      end
      $ 545 "Wait: 0.3"
      sleep(0.3)
      $ 546 "Set CO[1]=Encender"
      set_configurable_digital_out(1, True)
      $ 547 "Wait: 0.3"
      sleep(0.3)
      $ 548 "Loop 1 times"
      Loop_85 = 0
      while (Loop_85 < 1):
        $ 549 "bajar≔pose_add(get_actual_tcp_pose(), bajada_broca)"
        global bajar= pose_add ( get_actual_tcp_pose (), bajada_broca)
        $ 550 "bajar" "breakAfter"
        movel(bajar, a=0.005, v=0.001)
        $ 551 "subir≔pose_sub(get_actual_tcp_pose(), bajada_broca)"
        global subir= pose_sub ( get_actual_tcp_pose (), bajada_broca)
        $ 552 "subir" "breakAfter"
        movel(subir, a=0.01, v=0.005)
        $ 553 "bajada_broca≔pose_sub(bajada_broca, bajada)"
        global bajada_broca= pose_sub (bajada_broca, bajada)
        Loop_85 = Loop_85 + 1
      end
      $ 554 "Direction: Base Z+"
      global move_thread_flag_554=0
      thread move_thread_554():
        enter_critical
        move_thread_flag_554 = 1
        local towardsPos=calculate_point_to_move_towards(p[0.0,0.0,0.0,0.0,0.0,0.0], [0.0,0.0,1.0], 0.06)
        movel(towardsPos, a=0.035, v=0.03)
        move_thread_flag_554 = 2
        exit_critical
      end
      move_thread_flag_554 = 0
      move_thread_han_554 = run move_thread_554()
      while (True):
        sleep(1.0E-10)
        if (move_thread_flag_554 > 1):
          join move_thread_han_554
          $ 555 "Until (distance)"
          break
        end
        sync()
      end
      $ 556 "Set CO[1]=Apagar"
      set_configurable_digital_out(1, False)
      $ 557 "barreno_actual≔barreno_actual+1"
      global barreno_actual=barreno_actual+1
      $ 558 "Call Quitar_broca"
      Quitar_broca()
      $ 559 "Call Poner_broca"
      Poner_broca()
    end
    $ 560 "EF"
    $ 561 "'desbaste_inicial'"
    # 'desbaste_inicial'
    $ 562 "bajada_broca≔p[0,0,-0.012,0,0,0]"
    global bajada_broca=p[0,0,-0.012,0,0,0]
    $ 563 "barrenos_menos1≔8"
    global barrenos_menos1=8
    $ 564 "barreno_actual≔0"
    global barreno_actual=0
    $ 565 "Loop barreno_actual≤barrenos_menos1"
    while (barreno_actual <= barrenos_menos1):
      $ 566 "Perforacion"
      $ 567 "MoveL"
      $ 568 "internos≔interpolate_pose(Linea1_E, Linea1_F, barreno_actual/barrenos_menos1)"
      global internos= interpolate_pose (Linea1_E_p, Linea1_F_p, barreno_actual/barrenos_menos1)
      $ 569 "internos" "breakAfter"
      movel(internos, a=0.5, v=0.1)
      $ 570 "'desbaste_inicial'"
      # 'desbaste_inicial'
      $ 571 "bajada_broca≔p[0,0,-0.026,0,0,0]"
      global bajada_broca=p[0,0,-0.026,0,0,0]
      $ 572 "bajada≔p[0,0,0.026,0,0,0]"
      global bajada=p[0,0,0.026,0,0,0]
      $ 573 "Direction: Base Z-"
      global move_thread_flag_573=0
      thread move_thread_573():
        enter_critical
        move_thread_flag_573 = 1
        local towardsPos=calculate_point_to_move_towards(p[0.0,0.0,0.0,0.0,0.0,0.0], [0.0,0.0,-1.0], 0.08270000000000001)
        movel(towardsPos, a=0.015, v=0.015)
        move_thread_flag_573 = 2
        exit_critical
      end
      move_thread_flag_573 = 0
      move_thread_han_573 = run move_thread_573()
      while (True):
        sleep(1.0E-10)
        if (move_thread_flag_573 > 1):
          join move_thread_han_573
          $ 574 "Until (distance)"
          break
        end
        sync()
      end
      $ 575 "Popup: punto contacto alanzdo"
      popup("punto contacto alanzdo", "Mensaje", False, False, blocking=True)
      $ 576 "Direction: Base Z+"
      global move_thread_flag_576=0
      thread move_thread_576():
        enter_critical
        move_thread_flag_576 = 1
        local towardsPos=calculate_point_to_move_towards(p[0.0,0.0,0.0,0.0,0.0,0.0], [0.0,0.0,1.0], 0.002)
        movel(towardsPos, a=0.005, v=0.003)
        move_thread_flag_576 = 2
        exit_critical
      end
      move_thread_flag_576 = 0
      move_thread_han_576 = run move_thread_576()
      while (True):
        sleep(1.0E-10)
        if (move_thread_flag_576 > 1):
          join move_thread_han_576
          $ 577 "Until (distance)"
          break
        end
        sync()
      end
      $ 578 "Wait: 0.3"
      sleep(0.3)
      $ 579 "Set CO[1]=Encender"
      set_configurable_digital_out(1, True)
      $ 580 "Wait: 0.3"
      sleep(0.3)
      $ 581 "Loop 1 times"
      Loop_87 = 0
      while (Loop_87 < 1):
        $ 582 "bajar≔pose_add(get_actual_tcp_pose(), bajada_broca)"
        global bajar= pose_add ( get_actual_tcp_pose (), bajada_broca)
        $ 583 "bajar" "breakAfter"
        movel(bajar, a=0.005, v=0.001)
        $ 584 "subir≔pose_sub(get_actual_tcp_pose(), bajada_broca)"
        global subir= pose_sub ( get_actual_tcp_pose (), bajada_broca)
        $ 585 "subir" "breakAfter"
        movel(subir, a=0.01, v=0.005)
        $ 586 "bajada_broca≔pose_sub(bajada_broca, bajada)"
        global bajada_broca= pose_sub (bajada_broca, bajada)
        Loop_87 = Loop_87 + 1
      end
      $ 587 "Direction: Base Z+"
      global move_thread_flag_587=0
      thread move_thread_587():
        enter_critical
        move_thread_flag_587 = 1
        local towardsPos=calculate_point_to_move_towards(p[0.0,0.0,0.0,0.0,0.0,0.0], [0.0,0.0,1.0], 0.06)
        movel(towardsPos, a=0.035, v=0.03)
        move_thread_flag_587 = 2
        exit_critical
      end
      move_thread_flag_587 = 0
      move_thread_han_587 = run move_thread_587()
      while (True):
        sleep(1.0E-10)
        if (move_thread_flag_587 > 1):
          join move_thread_han_587
          $ 588 "Until (distance)"
          break
        end
        sync()
      end
      $ 589 "Set CO[1]=Apagar"
      set_configurable_digital_out(1, False)
      $ 590 "barreno_actual≔barreno_actual+1"
      global barreno_actual=barreno_actual+1
      $ 591 "Call Quitar_broca"
      Quitar_broca()
      $ 592 "Call Poner_broca"
      Poner_broca()
    end
    $ 593 "Popup: Linea1 con full Terminada!"
    popup("Linea1 con full Terminada!", "Mensaje", False, False, blocking=True)
    $ 594 "Linea2"
    $ 595 "Marcar_puntos"
    $ 596 "MoveL"
    $ 597 "Home2" "breakAfter"
    movel(Home2_p, a=0.5, v=0.1)
    $ 598 "Linea2_A" "breakAfter"
    movel(Linea2_A_p, a=0.5, v=0.1)
    $ 599 "Linea2_B" "breakAfter"
    movel(Linea2_B_p, a=0.5, v=0.1)
    $ 600 "Linea2_C" "breakAfter"
    movel(Linea2_C_p, a=0.5, v=0.1)
    $ 601 "Linea2_D" "breakAfter"
    movel(Linea2_D_p, a=0.5, v=0.1)
    $ 602 "Linea2_E" "breakAfter"
    movel(Linea2_E_p, a=0.5, v=0.1)
    $ 603 "Linea2_F" "breakAfter"
    movel(Linea2_F_p, a=0.5, v=0.1)
    $ 604 "AB"
    $ 605 "'desbaste_inicial'"
    # 'desbaste_inicial'
    $ 606 "bajada_broca≔p[0,0,-0.012,0,0,0]"
    global bajada_broca=p[0,0,-0.012,0,0,0]
    $ 607 "barrenos_menos1≔8"
    global barrenos_menos1=8
    $ 608 "barreno_actual≔0"
    global barreno_actual=0
    $ 609 "Loop barreno_actual≤barrenos_menos1"
    while (barreno_actual <= barrenos_menos1):
      $ 610 "Perforacion"
      $ 611 "MoveL"
      $ 612 "internos≔interpolate_pose(Linea2_A, Linea2_B, barreno_actual/barrenos_menos1)"
      global internos= interpolate_pose (Linea2_A_p, Linea2_B_p, barreno_actual/barrenos_menos1)
      $ 613 "internos" "breakAfter"
      movel(internos, a=0.5, v=0.1)
      $ 614 "'desbaste_inicial'"
      # 'desbaste_inicial'
      $ 615 "bajada_broca≔p[0,0,-0.026,0,0,0]"
      global bajada_broca=p[0,0,-0.026,0,0,0]
      $ 616 "bajada≔p[0,0,0.026,0,0,0]"
      global bajada=p[0,0,0.026,0,0,0]
      $ 617 "Direction: Base Z-"
      global move_thread_flag_617=0
      thread move_thread_617():
        enter_critical
        move_thread_flag_617 = 1
        local towardsPos=calculate_point_to_move_towards(p[0.0,0.0,0.0,0.0,0.0,0.0], [0.0,0.0,-1.0], 0.08270000000000001)
        movel(towardsPos, a=0.015, v=0.015)
        move_thread_flag_617 = 2
        exit_critical
      end
      move_thread_flag_617 = 0
      move_thread_han_617 = run move_thread_617()
      while (True):
        sleep(1.0E-10)
        if (move_thread_flag_617 > 1):
          join move_thread_han_617
          $ 618 "Until (distance)"
          break
        end
        sync()
      end
      $ 619 "Popup: punto contacto alanzdo"
      popup("punto contacto alanzdo", "Mensaje", False, False, blocking=True)
      $ 620 "Direction: Base Z+"
      global move_thread_flag_620=0
      thread move_thread_620():
        enter_critical
        move_thread_flag_620 = 1
        local towardsPos=calculate_point_to_move_towards(p[0.0,0.0,0.0,0.0,0.0,0.0], [0.0,0.0,1.0], 0.002)
        movel(towardsPos, a=0.005, v=0.003)
        move_thread_flag_620 = 2
        exit_critical
      end
      move_thread_flag_620 = 0
      move_thread_han_620 = run move_thread_620()
      while (True):
        sleep(1.0E-10)
        if (move_thread_flag_620 > 1):
          join move_thread_han_620
          $ 621 "Until (distance)"
          break
        end
        sync()
      end
      $ 622 "Wait: 0.3"
      sleep(0.3)
      $ 623 "Set CO[1]=Encender"
      set_configurable_digital_out(1, True)
      $ 624 "Wait: 0.3"
      sleep(0.3)
      $ 625 "Loop 1 times"
      Loop_90 = 0
      while (Loop_90 < 1):
        $ 626 "bajar≔pose_add(get_actual_tcp_pose(), bajada_broca)"
        global bajar= pose_add ( get_actual_tcp_pose (), bajada_broca)
        $ 627 "bajar" "breakAfter"
        movel(bajar, a=0.005, v=0.001)
        $ 628 "subir≔pose_sub(get_actual_tcp_pose(), bajada_broca)"
        global subir= pose_sub ( get_actual_tcp_pose (), bajada_broca)
        $ 629 "subir" "breakAfter"
        movel(subir, a=0.01, v=0.005)
        $ 630 "bajada_broca≔pose_sub(bajada_broca, bajada)"
        global bajada_broca= pose_sub (bajada_broca, bajada)
        Loop_90 = Loop_90 + 1
      end
      $ 631 "Direction: Base Z+"
      global move_thread_flag_631=0
      thread move_thread_631():
        enter_critical
        move_thread_flag_631 = 1
        local towardsPos=calculate_point_to_move_towards(p[0.0,0.0,0.0,0.0,0.0,0.0], [0.0,0.0,1.0], 0.06)
        movel(towardsPos, a=0.035, v=0.03)
        move_thread_flag_631 = 2
        exit_critical
      end
      move_thread_flag_631 = 0
      move_thread_han_631 = run move_thread_631()
      while (True):
        sleep(1.0E-10)
        if (move_thread_flag_631 > 1):
          join move_thread_han_631
          $ 632 "Until (distance)"
          break
        end
        sync()
      end
      $ 633 "Set CO[1]=Apagar"
      set_configurable_digital_out(1, False)
      $ 634 "barreno_actual≔barreno_actual+1"
      global barreno_actual=barreno_actual+1
      $ 635 "Call Quitar_broca"
      Quitar_broca()
      $ 636 "Call Poner_broca"
      Poner_broca()
    end
    $ 637 "CD"
    $ 638 "'desbaste_inicial'"
    # 'desbaste_inicial'
    $ 639 "bajada_broca≔p[0,0,-0.012,0,0,0]"
    global bajada_broca=p[0,0,-0.012,0,0,0]
    $ 640 "barrenos_menos1≔8"
    global barrenos_menos1=8
    $ 641 "barreno_actual≔0"
    global barreno_actual=0
    $ 642 "Loop barreno_actual≤barrenos_menos1"
    while (barreno_actual <= barrenos_menos1):
      $ 643 "Perforacion"
      $ 644 "MoveL"
      $ 645 "internos≔interpolate_pose(Linea2_C, Linea2_D, barreno_actual/barrenos_menos1)"
      global internos= interpolate_pose (Linea2_C_p, Linea2_D_p, barreno_actual/barrenos_menos1)
      $ 646 "internos" "breakAfter"
      movel(internos, a=0.5, v=0.1)
      $ 647 "'desbaste_inicial'"
      # 'desbaste_inicial'
      $ 648 "bajada_broca≔p[0,0,-0.026,0,0,0]"
      global bajada_broca=p[0,0,-0.026,0,0,0]
      $ 649 "bajada≔p[0,0,0.026,0,0,0]"
      global bajada=p[0,0,0.026,0,0,0]
      $ 650 "Direction: Base Z-"
      global move_thread_flag_650=0
      thread move_thread_650():
        enter_critical
        move_thread_flag_650 = 1
        local towardsPos=calculate_point_to_move_towards(p[0.0,0.0,0.0,0.0,0.0,0.0], [0.0,0.0,-1.0], 0.08270000000000001)
        movel(towardsPos, a=0.015, v=0.015)
        move_thread_flag_650 = 2
        exit_critical
      end
      move_thread_flag_650 = 0
      move_thread_han_650 = run move_thread_650()
      while (True):
        sleep(1.0E-10)
        if (move_thread_flag_650 > 1):
          join move_thread_han_650
          $ 651 "Until (distance)"
          break
        end
        sync()
      end
      $ 652 "Popup: punto contacto alanzdo"
      popup("punto contacto alanzdo", "Mensaje", False, False, blocking=True)
      $ 653 "Direction: Base Z+"
      global move_thread_flag_653=0
      thread move_thread_653():
        enter_critical
        move_thread_flag_653 = 1
        local towardsPos=calculate_point_to_move_towards(p[0.0,0.0,0.0,0.0,0.0,0.0], [0.0,0.0,1.0], 0.002)
        movel(towardsPos, a=0.005, v=0.003)
        move_thread_flag_653 = 2
        exit_critical
      end
      move_thread_flag_653 = 0
      move_thread_han_653 = run move_thread_653()
      while (True):
        sleep(1.0E-10)
        if (move_thread_flag_653 > 1):
          join move_thread_han_653
          $ 654 "Until (distance)"
          break
        end
        sync()
      end
      $ 655 "Wait: 0.3"
      sleep(0.3)
      $ 656 "Set CO[1]=Encender"
      set_configurable_digital_out(1, True)
      $ 657 "Wait: 0.3"
      sleep(0.3)
      $ 658 "Loop 1 times"
      Loop_92 = 0
      while (Loop_92 < 1):
        $ 659 "bajar≔pose_add(get_actual_tcp_pose(), bajada_broca)"
        global bajar= pose_add ( get_actual_tcp_pose (), bajada_broca)
        $ 660 "bajar" "breakAfter"
        movel(bajar, a=0.005, v=0.001)
        $ 661 "subir≔pose_sub(get_actual_tcp_pose(), bajada_broca)"
        global subir= pose_sub ( get_actual_tcp_pose (), bajada_broca)
        $ 662 "subir" "breakAfter"
        movel(subir, a=0.01, v=0.005)
        $ 663 "bajada_broca≔pose_sub(bajada_broca, bajada)"
        global bajada_broca= pose_sub (bajada_broca, bajada)
        Loop_92 = Loop_92 + 1
      end
      $ 664 "Direction: Base Z+"
      global move_thread_flag_664=0
      thread move_thread_664():
        enter_critical
        move_thread_flag_664 = 1
        local towardsPos=calculate_point_to_move_towards(p[0.0,0.0,0.0,0.0,0.0,0.0], [0.0,0.0,1.0], 0.06)
        movel(towardsPos, a=0.035, v=0.03)
        move_thread_flag_664 = 2
        exit_critical
      end
      move_thread_flag_664 = 0
      move_thread_han_664 = run move_thread_664()
      while (True):
        sleep(1.0E-10)
        if (move_thread_flag_664 > 1):
          join move_thread_han_664
          $ 665 "Until (distance)"
          break
        end
        sync()
      end
      $ 666 "Set CO[1]=Apagar"
      set_configurable_digital_out(1, False)
      $ 667 "barreno_actual≔barreno_actual+1"
      global barreno_actual=barreno_actual+1
      $ 668 "Call Quitar_broca"
      Quitar_broca()
      $ 669 "Call Poner_broca"
      Poner_broca()
    end
    $ 670 "EF"
    $ 671 "'desbaste_inicial'"
    # 'desbaste_inicial'
    $ 672 "bajada_broca≔p[0,0,-0.012,0,0,0]"
    global bajada_broca=p[0,0,-0.012,0,0,0]
    $ 673 "barrenos_menos1≔8"
    global barrenos_menos1=8
    $ 674 "barreno_actual≔0"
    global barreno_actual=0
    $ 675 "Loop barreno_actual≤barrenos_menos1"
    while (barreno_actual <= barrenos_menos1):
      $ 676 "Perforacion"
      $ 677 "MoveL"
      $ 678 "internos≔interpolate_pose(Linea2_E, Linea2_F, barreno_actual/barrenos_menos1)"
      global internos= interpolate_pose (Linea2_E_p, Linea2_F_p, barreno_actual/barrenos_menos1)
      $ 679 "internos" "breakAfter"
      movel(internos, a=0.5, v=0.1)
      $ 680 "'desbaste_inicial'"
      # 'desbaste_inicial'
      $ 681 "bajada_broca≔p[0,0,-0.026,0,0,0]"
      global bajada_broca=p[0,0,-0.026,0,0,0]
      $ 682 "bajada≔p[0,0,0.026,0,0,0]"
      global bajada=p[0,0,0.026,0,0,0]
      $ 683 "Direction: Base Z-"
      global move_thread_flag_683=0
      thread move_thread_683():
        enter_critical
        move_thread_flag_683 = 1
        local towardsPos=calculate_point_to_move_towards(p[0.0,0.0,0.0,0.0,0.0,0.0], [0.0,0.0,-1.0], 0.08270000000000001)
        movel(towardsPos, a=0.015, v=0.015)
        move_thread_flag_683 = 2
        exit_critical
      end
      move_thread_flag_683 = 0
      move_thread_han_683 = run move_thread_683()
      while (True):
        sleep(1.0E-10)
        if (move_thread_flag_683 > 1):
          join move_thread_han_683
          $ 684 "Until (distance)"
          break
        end
        sync()
      end
      $ 685 "Popup: punto contacto alanzdo"
      popup("punto contacto alanzdo", "Mensaje", False, False, blocking=True)
      $ 686 "Direction: Base Z+"
      global move_thread_flag_686=0
      thread move_thread_686():
        enter_critical
        move_thread_flag_686 = 1
        local towardsPos=calculate_point_to_move_towards(p[0.0,0.0,0.0,0.0,0.0,0.0], [0.0,0.0,1.0], 0.002)
        movel(towardsPos, a=0.005, v=0.003)
        move_thread_flag_686 = 2
        exit_critical
      end
      move_thread_flag_686 = 0
      move_thread_han_686 = run move_thread_686()
      while (True):
        sleep(1.0E-10)
        if (move_thread_flag_686 > 1):
          join move_thread_han_686
          $ 687 "Until (distance)"
          break
        end
        sync()
      end
      $ 688 "Wait: 0.3"
      sleep(0.3)
      $ 689 "Set CO[1]=Encender"
      set_configurable_digital_out(1, True)
      $ 690 "Wait: 0.3"
      sleep(0.3)
      $ 691 "Loop 1 times"
      Loop_94 = 0
      while (Loop_94 < 1):
        $ 692 "bajar≔pose_add(get_actual_tcp_pose(), bajada_broca)"
        global bajar= pose_add ( get_actual_tcp_pose (), bajada_broca)
        $ 693 "bajar" "breakAfter"
        movel(bajar, a=0.005, v=0.001)
        $ 694 "subir≔pose_sub(get_actual_tcp_pose(), bajada_broca)"
        global subir= pose_sub ( get_actual_tcp_pose (), bajada_broca)
        $ 695 "subir" "breakAfter"
        movel(subir, a=0.01, v=0.005)
        $ 696 "bajada_broca≔pose_sub(bajada_broca, bajada)"
        global bajada_broca= pose_sub (bajada_broca, bajada)
        Loop_94 = Loop_94 + 1
      end
      $ 697 "Direction: Base Z+"
      global move_thread_flag_697=0
      thread move_thread_697():
        enter_critical
        move_thread_flag_697 = 1
        local towardsPos=calculate_point_to_move_towards(p[0.0,0.0,0.0,0.0,0.0,0.0], [0.0,0.0,1.0], 0.06)
        movel(towardsPos, a=0.035, v=0.03)
        move_thread_flag_697 = 2
        exit_critical
      end
      move_thread_flag_697 = 0
      move_thread_han_697 = run move_thread_697()
      while (True):
        sleep(1.0E-10)
        if (move_thread_flag_697 > 1):
          join move_thread_han_697
          $ 698 "Until (distance)"
          break
        end
        sync()
      end
      $ 699 "Set CO[1]=Apagar"
      set_configurable_digital_out(1, False)
      $ 700 "barreno_actual≔barreno_actual+1"
      global barreno_actual=barreno_actual+1
      $ 701 "If barreno_actual≥barrenos_menos1"
      if (barreno_actual >= barrenos_menos1):
        $ 702 "cambiar_broca≔ True "
        global cambiar_broca=  True
      end
      $ 703 "Call Quitar_broca"
      Quitar_broca()
      $ 704 "Call Poner_broca"
      Poner_broca()
    end
    $ 705 "Popup: Linea2 con full Terminada!"
    popup("Linea2 con full Terminada!", "Mensaje", False, False, blocking=True)
    $ 706 "600"
    $ 1218 "Broca_1"
    $ 1219 "Linea7"
    $ 1220 "Marcar_puntos"
    $ 1221 "MoveL"
    $ 1222 "Home2" "breakAfter"
    movel(Home2_p, a=0.5, v=0.1)
    $ 1223 "Linea7_A" "breakAfter"
    movel(Linea7_A_p, a=0.5, v=0.1)
    $ 1224 "bajada_comprobacion"
    $ 1225 "Direction: Base Z-"
    global move_thread_flag_1225=0
    thread move_thread_1225():
      enter_critical
      move_thread_flag_1225 = 1
      local towardsPos=calculate_point_to_move_towards(p[0.0,0.0,0.0,0.0,0.0,0.0], [0.0,0.0,-1.0], 0.071)
      movel(towardsPos, a=0.15, v=0.1)
      move_thread_flag_1225 = 2
      exit_critical
    end
    move_thread_flag_1225 = 0
    move_thread_han_1225 = run move_thread_1225()
    while (True):
      sleep(1.0E-10)
      if (move_thread_flag_1225 > 1):
        join move_thread_han_1225
        $ 1226 "Until (distance)"
        break
      end
      sync()
    end
    $ 1227 "Direction: Base Z-"
    global move_thread_flag_1227=0
    thread move_thread_1227():
      enter_critical
      move_thread_flag_1227 = 1
      local towardsPos=calculate_point_to_move_towards(p[0.0,0.0,0.0,0.0,0.0,0.0], [0.0,0.0,-1.0], 1000.0)
      movel(towardsPos, a=0.007, v=0.007)
      move_thread_flag_1227 = 2
      exit_critical
    end
    move_thread_flag_1227 = 0
    move_thread_han_1227 = run move_thread_1227()
    while (True):
      local targetTcpDirection=get_target_tcp_speed()
      local stepsToRetract=tool_contact(direction=targetTcpDirection)
      if (stepsToRetract > 0):
        kill move_thread_han_1227
        stopl(0.02)
        local backTrackMovement=get_actual_joint_positions_history(stepsToRetract)
        local contactPose=get_forward_kin(backTrackMovement)
        local posDir=[targetTcpDirection[0],targetTcpDirection[1],targetTcpDirection[2]]
        local retractTo=contactPose
        if (norm(posDir) > 1e-6):
          local normalizedPosDir=normalize(posDir)
          local additionalRetraction=p[normalizedPosDir[0] * 0.0, normalizedPosDir[1] * 0.0, normalizedPosDir[2] * 0.0, 0, 0, 0]
          retractTo = pose_sub(contactPose, additionalRetraction)
        end
        movel(retractTo, a=0.02, v=0.1)
        $ 1228 "Until (tool_contact_detection)"
        break
      end
      sync()
    end
    $ 1229 "Direction: Base Z+"
    global move_thread_flag_1229=0
    thread move_thread_1229():
      enter_critical
      move_thread_flag_1229 = 1
      local towardsPos=calculate_point_to_move_towards(p[0.0,0.0,0.0,0.0,0.0,0.0], [0.0,0.0,1.0], 0.08)
      movel(towardsPos, a=0.15, v=0.1)
      move_thread_flag_1229 = 2
      exit_critical
    end
    move_thread_flag_1229 = 0
    move_thread_han_1229 = run move_thread_1229()
    while (True):
      sleep(1.0E-10)
      if (move_thread_flag_1229 > 1):
        join move_thread_han_1229
        $ 1230 "Until (distance)"
        break
      end
      sync()
    end
    $ 1231 "Linea7_B" "breakAfter"
    movel(Linea7_B_p, a=0.5, v=0.1)
    $ 1232 "bajada_comprobacion"
    $ 1233 "Direction: Base Z-"
    global move_thread_flag_1233=0
    thread move_thread_1233():
      enter_critical
      move_thread_flag_1233 = 1
      local towardsPos=calculate_point_to_move_towards(p[0.0,0.0,0.0,0.0,0.0,0.0], [0.0,0.0,-1.0], 0.071)
      movel(towardsPos, a=0.15, v=0.1)
      move_thread_flag_1233 = 2
      exit_critical
    end
    move_thread_flag_1233 = 0
    move_thread_han_1233 = run move_thread_1233()
    while (True):
      sleep(1.0E-10)
      if (move_thread_flag_1233 > 1):
        join move_thread_han_1233
        $ 1234 "Until (distance)"
        break
      end
      sync()
    end
    $ 1235 "Direction: Base Z-"
    global move_thread_flag_1235=0
    thread move_thread_1235():
      enter_critical
      move_thread_flag_1235 = 1
      local towardsPos=calculate_point_to_move_towards(p[0.0,0.0,0.0,0.0,0.0,0.0], [0.0,0.0,-1.0], 1000.0)
      movel(towardsPos, a=0.007, v=0.007)
      move_thread_flag_1235 = 2
      exit_critical
    end
    move_thread_flag_1235 = 0
    move_thread_han_1235 = run move_thread_1235()
    while (True):
      local targetTcpDirection=get_target_tcp_speed()
      local stepsToRetract=tool_contact(direction=targetTcpDirection)
      if (stepsToRetract > 0):
        kill move_thread_han_1235
        stopl(0.02)
        local backTrackMovement=get_actual_joint_positions_history(stepsToRetract)
        local contactPose=get_forward_kin(backTrackMovement)
        local posDir=[targetTcpDirection[0],targetTcpDirection[1],targetTcpDirection[2]]
        local retractTo=contactPose
        if (norm(posDir) > 1e-6):
          local normalizedPosDir=normalize(posDir)
          local additionalRetraction=p[normalizedPosDir[0] * 0.0, normalizedPosDir[1] * 0.0, normalizedPosDir[2] * 0.0, 0, 0, 0]
          retractTo = pose_sub(contactPose, additionalRetraction)
        end
        movel(retractTo, a=0.02, v=0.1)
        $ 1236 "Until (tool_contact_detection)"
        break
      end
      sync()
    end
    $ 1237 "Direction: Base Z+"
    global move_thread_flag_1237=0
    thread move_thread_1237():
      enter_critical
      move_thread_flag_1237 = 1
      local towardsPos=calculate_point_to_move_towards(p[0.0,0.0,0.0,0.0,0.0,0.0], [0.0,0.0,1.0], 0.08)
      movel(towardsPos, a=0.15, v=0.1)
      move_thread_flag_1237 = 2
      exit_critical
    end
    move_thread_flag_1237 = 0
    move_thread_han_1237 = run move_thread_1237()
    while (True):
      sleep(1.0E-10)
      if (move_thread_flag_1237 > 1):
        join move_thread_han_1237
        $ 1238 "Until (distance)"
        break
      end
      sync()
    end
    $ 1239 "AB"
    $ 1240 "'desbaste_inicial'"
    # 'desbaste_inicial'
    $ 1241 "bajada_broca≔p[0,0,-0.008,0,0,0]"
    global bajada_broca=p[0,0,-0.008,0,0,0]
    $ 1242 "barrenos_menos1≔2"
    global barrenos_menos1=2
    $ 1243 "barreno_actual≔1"
    global barreno_actual=1
    $ 1244 "Loop barreno_actual≤barrenos_menos1"
    while (barreno_actual <= barrenos_menos1):
      $ 1245 "Perforacion"
      $ 1246 "MoveL"
      $ 1247 "internos≔interpolate_pose(Linea7_A, Linea7_B, barreno_actual/barrenos_menos1)"
      global internos= interpolate_pose (Linea7_A_p, Linea7_B_p, barreno_actual/barrenos_menos1)
      $ 1248 "internos" "breakAfter"
      movel(internos, a=0.5, v=0.1)
      $ 1249 "'desbaste_inicial'"
      # 'desbaste_inicial'
      $ 1250 "bajada_broca≔p[0,0,-0.024,0,0,0]"
      global bajada_broca=p[0,0,-0.024,0,0,0]
      $ 1251 "bajada≔p[0,0,0.024,0,0,0]"
      global bajada=p[0,0,0.024,0,0,0]
      $ 1252 "Direction: Base Z-"
      global move_thread_flag_1252=0
      thread move_thread_1252():
        enter_critical
        move_thread_flag_1252 = 1
        local towardsPos=calculate_point_to_move_towards(p[0.0,0.0,0.0,0.0,0.0,0.0], [0.0,0.0,-1.0], 0.071)
        movel(towardsPos, a=0.15, v=0.1)
        move_thread_flag_1252 = 2
        exit_critical
      end
      move_thread_flag_1252 = 0
      move_thread_han_1252 = run move_thread_1252()
      while (True):
        sleep(1.0E-10)
        if (move_thread_flag_1252 > 1):
          join move_thread_han_1252
          $ 1253 "Until (distance)"
          break
        end
        sync()
      end
      $ 1254 "Direction: Base Z-"
      global move_thread_flag_1254=0
      thread move_thread_1254():
        enter_critical
        move_thread_flag_1254 = 1
        local towardsPos=calculate_point_to_move_towards(p[0.0,0.0,0.0,0.0,0.0,0.0], [0.0,0.0,-1.0], 1000.0)
        movel(towardsPos, a=0.007, v=0.007)
        move_thread_flag_1254 = 2
        exit_critical
      end
      move_thread_flag_1254 = 0
      move_thread_han_1254 = run move_thread_1254()
      while (True):
        local targetTcpDirection=get_target_tcp_speed()
        local stepsToRetract=tool_contact(direction=targetTcpDirection)
        if (stepsToRetract > 0):
          kill move_thread_han_1254
          stopl(0.02)
          local backTrackMovement=get_actual_joint_positions_history(stepsToRetract)
          local contactPose=get_forward_kin(backTrackMovement)
          local posDir=[targetTcpDirection[0],targetTcpDirection[1],targetTcpDirection[2]]
          local retractTo=contactPose
          if (norm(posDir) > 1e-6):
            local normalizedPosDir=normalize(posDir)
            local additionalRetraction=p[normalizedPosDir[0] * 0.0, normalizedPosDir[1] * 0.0, normalizedPosDir[2] * 0.0, 0, 0, 0]
            retractTo = pose_sub(contactPose, additionalRetraction)
          end
          movel(retractTo, a=0.02, v=0.1)
          $ 1255 "Until (tool_contact_detection)"
          break
        end
        sync()
      end
      $ 1256 "Popup: punto contacto alanzdo"
      popup("punto contacto alanzdo", "Mensaje", False, False, blocking=True)
      $ 1257 "Direction: Base Z+"
      global move_thread_flag_1257=0
      thread move_thread_1257():
        enter_critical
        move_thread_flag_1257 = 1
        local towardsPos=calculate_point_to_move_towards(p[0.0,0.0,0.0,0.0,0.0,0.0], [0.0,0.0,1.0], 0.007)
        movel(towardsPos, a=0.015, v=0.015)
        move_thread_flag_1257 = 2
        exit_critical
      end
      move_thread_flag_1257 = 0
      move_thread_han_1257 = run move_thread_1257()
      while (True):
        sleep(1.0E-10)
        if (move_thread_flag_1257 > 1):
          join move_thread_han_1257
          $ 1258 "Until (distance)"
          break
        end
        sync()
      end
      $ 1259 "Wait: 0.3"
      sleep(0.3)
      $ 1260 "Set CO[1]=Encender"
      set_configurable_digital_out(1, True)
      $ 1261 "Wait: 0.3"
      sleep(0.3)
      $ 1262 "Loop 1 times"
      Loop_96 = 0
      while (Loop_96 < 1):
        $ 1263 "bajar≔pose_add(get_actual_tcp_pose(), bajada_broca)"
        global bajar= pose_add ( get_actual_tcp_pose (), bajada_broca)
        $ 1264 "bajar" "breakAfter"
        movel(bajar, a=0.004, v=0.004)
        $ 1265 "subir≔pose_sub(get_actual_tcp_pose(), bajada_broca)"
        global subir= pose_sub ( get_actual_tcp_pose (), bajada_broca)
        $ 1266 "Direction: Base Z+"
        global move_thread_flag_1266=0
        thread move_thread_1266():
          enter_critical
          move_thread_flag_1266 = 1
          local towardsPos=calculate_point_to_move_towards(p[0.0,0.0,0.0,0.0,0.0,0.0], [0.0,0.0,1.0], 0.002)
          movel(towardsPos, a=0.015, v=0.015)
          move_thread_flag_1266 = 2
          exit_critical
        end
        move_thread_flag_1266 = 0
        move_thread_han_1266 = run move_thread_1266()
        while (True):
          sleep(1.0E-10)
          if (move_thread_flag_1266 > 1):
            join move_thread_han_1266
            $ 1267 "Until (distance)"
            break
          end
          sync()
        end
        $ 1268 "Set CO[1]=Apagar"
        set_configurable_digital_out(1, False)
        $ 1269 "subir" "breakAfter"
        movel(subir, a=0.015, v=0.015)
        $ 1270 "bajada_broca≔pose_sub(bajada_broca, bajada)"
        global bajada_broca= pose_sub (bajada_broca, bajada)
        Loop_96 = Loop_96 + 1
      end
      $ 1271 "Direction: Base Z+"
      global move_thread_flag_1271=0
      thread move_thread_1271():
        enter_critical
        move_thread_flag_1271 = 1
        local towardsPos=calculate_point_to_move_towards(p[0.0,0.0,0.0,0.0,0.0,0.0], [0.0,0.0,1.0], 0.08)
        movel(towardsPos, a=0.15, v=0.1)
        move_thread_flag_1271 = 2
        exit_critical
      end
      move_thread_flag_1271 = 0
      move_thread_han_1271 = run move_thread_1271()
      while (True):
        sleep(1.0E-10)
        if (move_thread_flag_1271 > 1):
          join move_thread_han_1271
          $ 1272 "Until (distance)"
          break
        end
        sync()
      end
      $ 1273 "Set CO[1]=Apagar"
      set_configurable_digital_out(1, False)
      $ 1274 "barreno_actual≔barreno_actual+1"
      global barreno_actual=barreno_actual+1
      $ 1275 "Call Quitar_broca"
      Quitar_broca()
      $ 1276 "Call Poner_broca"
      Poner_broca()
    end
    $ 1277 "Popup: Linea7 con chica Terminada!"
    popup("Linea7 con chica Terminada!", "Mensaje", False, False, blocking=True)
    $ 1278 "Linea8"
    $ 1279 "Marcar_puntos"
    $ 1280 "MoveL"
    $ 1281 "Linea8_A" "breakAfter"
    movel(Linea8_A_p, a=0.5, v=0.1)
    $ 1282 "bajada_comprobacion"
    $ 1283 "Direction: Base Z-"
    global move_thread_flag_1283=0
    thread move_thread_1283():
      enter_critical
      move_thread_flag_1283 = 1
      local towardsPos=calculate_point_to_move_towards(p[0.0,0.0,0.0,0.0,0.0,0.0], [0.0,0.0,-1.0], 0.071)
      movel(towardsPos, a=0.15, v=0.1)
      move_thread_flag_1283 = 2
      exit_critical
    end
    move_thread_flag_1283 = 0
    move_thread_han_1283 = run move_thread_1283()
    while (True):
      sleep(1.0E-10)
      if (move_thread_flag_1283 > 1):
        join move_thread_han_1283
        $ 1284 "Until (distance)"
        break
      end
      sync()
    end
    $ 1285 "Direction: Base Z-"
    global move_thread_flag_1285=0
    thread move_thread_1285():
      enter_critical
      move_thread_flag_1285 = 1
      local towardsPos=calculate_point_to_move_towards(p[0.0,0.0,0.0,0.0,0.0,0.0], [0.0,0.0,-1.0], 1000.0)
      movel(towardsPos, a=0.007, v=0.007)
      move_thread_flag_1285 = 2
      exit_critical
    end
    move_thread_flag_1285 = 0
    move_thread_han_1285 = run move_thread_1285()
    while (True):
      local targetTcpDirection=get_target_tcp_speed()
      local stepsToRetract=tool_contact(direction=targetTcpDirection)
      if (stepsToRetract > 0):
        kill move_thread_han_1285
        stopl(0.02)
        local backTrackMovement=get_actual_joint_positions_history(stepsToRetract)
        local contactPose=get_forward_kin(backTrackMovement)
        local posDir=[targetTcpDirection[0],targetTcpDirection[1],targetTcpDirection[2]]
        local retractTo=contactPose
        if (norm(posDir) > 1e-6):
          local normalizedPosDir=normalize(posDir)
          local additionalRetraction=p[normalizedPosDir[0] * 0.0, normalizedPosDir[1] * 0.0, normalizedPosDir[2] * 0.0, 0, 0, 0]
          retractTo = pose_sub(contactPose, additionalRetraction)
        end
        movel(retractTo, a=0.02, v=0.1)
        $ 1286 "Until (tool_contact_detection)"
        break
      end
      sync()
    end
    $ 1287 "Direction: Base Z+"
    global move_thread_flag_1287=0
    thread move_thread_1287():
      enter_critical
      move_thread_flag_1287 = 1
      local towardsPos=calculate_point_to_move_towards(p[0.0,0.0,0.0,0.0,0.0,0.0], [0.0,0.0,1.0], 0.08)
      movel(towardsPos, a=0.15, v=0.1)
      move_thread_flag_1287 = 2
      exit_critical
    end
    move_thread_flag_1287 = 0
    move_thread_han_1287 = run move_thread_1287()
    while (True):
      sleep(1.0E-10)
      if (move_thread_flag_1287 > 1):
        join move_thread_han_1287
        $ 1288 "Until (distance)"
        break
      end
      sync()
    end
    $ 1289 "Linea8_B" "breakAfter"
    movel(Linea8_B_p, a=0.5, v=0.1)
    $ 1290 "bajada_comprobacion"
    $ 1291 "Direction: Base Z-"
    global move_thread_flag_1291=0
    thread move_thread_1291():
      enter_critical
      move_thread_flag_1291 = 1
      local towardsPos=calculate_point_to_move_towards(p[0.0,0.0,0.0,0.0,0.0,0.0], [0.0,0.0,-1.0], 0.071)
      movel(towardsPos, a=0.15, v=0.1)
      move_thread_flag_1291 = 2
      exit_critical
    end
    move_thread_flag_1291 = 0
    move_thread_han_1291 = run move_thread_1291()
    while (True):
      sleep(1.0E-10)
      if (move_thread_flag_1291 > 1):
        join move_thread_han_1291
        $ 1292 "Until (distance)"
        break
      end
      sync()
    end
    $ 1293 "Direction: Base Z-"
    global move_thread_flag_1293=0
    thread move_thread_1293():
      enter_critical
      move_thread_flag_1293 = 1
      local towardsPos=calculate_point_to_move_towards(p[0.0,0.0,0.0,0.0,0.0,0.0], [0.0,0.0,-1.0], 1000.0)
      movel(towardsPos, a=0.007, v=0.007)
      move_thread_flag_1293 = 2
      exit_critical
    end
    move_thread_flag_1293 = 0
    move_thread_han_1293 = run move_thread_1293()
    while (True):
      local targetTcpDirection=get_target_tcp_speed()
      local stepsToRetract=tool_contact(direction=targetTcpDirection)
      if (stepsToRetract > 0):
        kill move_thread_han_1293
        stopl(0.02)
        local backTrackMovement=get_actual_joint_positions_history(stepsToRetract)
        local contactPose=get_forward_kin(backTrackMovement)
        local posDir=[targetTcpDirection[0],targetTcpDirection[1],targetTcpDirection[2]]
        local retractTo=contactPose
        if (norm(posDir) > 1e-6):
          local normalizedPosDir=normalize(posDir)
          local additionalRetraction=p[normalizedPosDir[0] * 0.0, normalizedPosDir[1] * 0.0, normalizedPosDir[2] * 0.0, 0, 0, 0]
          retractTo = pose_sub(contactPose, additionalRetraction)
        end
        movel(retractTo, a=0.02, v=0.1)
        $ 1294 "Until (tool_contact_detection)"
        break
      end
      sync()
    end
    $ 1295 "Direction: Base Z+"
    global move_thread_flag_1295=0
    thread move_thread_1295():
      enter_critical
      move_thread_flag_1295 = 1
      local towardsPos=calculate_point_to_move_towards(p[0.0,0.0,0.0,0.0,0.0,0.0], [0.0,0.0,1.0], 0.08)
      movel(towardsPos, a=0.15, v=0.1)
      move_thread_flag_1295 = 2
      exit_critical
    end
    move_thread_flag_1295 = 0
    move_thread_han_1295 = run move_thread_1295()
    while (True):
      sleep(1.0E-10)
      if (move_thread_flag_1295 > 1):
        join move_thread_han_1295
        $ 1296 "Until (distance)"
        break
      end
      sync()
    end
    $ 1297 "AB"
    $ 1298 "'desbaste_inicial'"
    # 'desbaste_inicial'
    $ 1299 "bajada_broca≔p[0,0,-0.008,0,0,0]"
    global bajada_broca=p[0,0,-0.008,0,0,0]
    $ 1300 "barrenos_menos1≔5"
    global barrenos_menos1=5
    $ 1301 "barreno_actual≔0"
    global barreno_actual=0
    $ 1302 "Loop barreno_actual≤barrenos_menos1"
    while (barreno_actual <= barrenos_menos1):
      $ 1303 "Perforacion"
      $ 1304 "MoveL"
      $ 1305 "internos≔interpolate_pose(Linea8_A, Linea8_B, barreno_actual/barrenos_menos1)"
      global internos= interpolate_pose (Linea8_A_p, Linea8_B_p, barreno_actual/barrenos_menos1)
      $ 1306 "internos" "breakAfter"
      movel(internos, a=0.5, v=0.1)
      $ 1307 "'desbaste_inicial'"
      # 'desbaste_inicial'
      $ 1308 "bajada_broca≔p[0,0,-0.024,0,0,0]"
      global bajada_broca=p[0,0,-0.024,0,0,0]
      $ 1309 "bajada≔p[0,0,0.0024,0,0,0]"
      global bajada=p[0,0,0.0024,0,0,0]
      $ 1310 "Direction: Base Z-"
      global move_thread_flag_1310=0
      thread move_thread_1310():
        enter_critical
        move_thread_flag_1310 = 1
        local towardsPos=calculate_point_to_move_towards(p[0.0,0.0,0.0,0.0,0.0,0.0], [0.0,0.0,-1.0], 0.071)
        movel(towardsPos, a=0.15, v=0.1)
        move_thread_flag_1310 = 2
        exit_critical
      end
      move_thread_flag_1310 = 0
      move_thread_han_1310 = run move_thread_1310()
      while (True):
        sleep(1.0E-10)
        if (move_thread_flag_1310 > 1):
          join move_thread_han_1310
          $ 1311 "Until (distance)"
          break
        end
        sync()
      end
      $ 1312 "Direction: Base Z-"
      global move_thread_flag_1312=0
      thread move_thread_1312():
        enter_critical
        move_thread_flag_1312 = 1
        local towardsPos=calculate_point_to_move_towards(p[0.0,0.0,0.0,0.0,0.0,0.0], [0.0,0.0,-1.0], 1000.0)
        movel(towardsPos, a=0.007, v=0.007)
        move_thread_flag_1312 = 2
        exit_critical
      end
      move_thread_flag_1312 = 0
      move_thread_han_1312 = run move_thread_1312()
      while (True):
        local targetTcpDirection=get_target_tcp_speed()
        local stepsToRetract=tool_contact(direction=targetTcpDirection)
        if (stepsToRetract > 0):
          kill move_thread_han_1312
          stopl(0.02)
          local backTrackMovement=get_actual_joint_positions_history(stepsToRetract)
          local contactPose=get_forward_kin(backTrackMovement)
          local posDir=[targetTcpDirection[0],targetTcpDirection[1],targetTcpDirection[2]]
          local retractTo=contactPose
          if (norm(posDir) > 1e-6):
            local normalizedPosDir=normalize(posDir)
            local additionalRetraction=p[normalizedPosDir[0] * 0.0, normalizedPosDir[1] * 0.0, normalizedPosDir[2] * 0.0, 0, 0, 0]
            retractTo = pose_sub(contactPose, additionalRetraction)
          end
          movel(retractTo, a=0.02, v=0.1)
          $ 1313 "Until (tool_contact_detection)"
          break
        end
        sync()
      end
      $ 1314 "Popup: punto contacto alanzdo"
      popup("punto contacto alanzdo", "Mensaje", False, False, blocking=True)
      $ 1315 "Direction: Base Z+"
      global move_thread_flag_1315=0
      thread move_thread_1315():
        enter_critical
        move_thread_flag_1315 = 1
        local towardsPos=calculate_point_to_move_towards(p[0.0,0.0,0.0,0.0,0.0,0.0], [0.0,0.0,1.0], 0.007)
        movel(towardsPos, a=0.015, v=0.015)
        move_thread_flag_1315 = 2
        exit_critical
      end
      move_thread_flag_1315 = 0
      move_thread_han_1315 = run move_thread_1315()
      while (True):
        sleep(1.0E-10)
        if (move_thread_flag_1315 > 1):
          join move_thread_han_1315
          $ 1316 "Until (distance)"
          break
        end
        sync()
      end
      $ 1317 "Wait: 0.3"
      sleep(0.3)
      $ 1318 "Set CO[1]=Encender"
      set_configurable_digital_out(1, True)
      $ 1319 "Wait: 0.3"
      sleep(0.3)
      $ 1320 "Loop 1 times"
      Loop_110 = 0
      while (Loop_110 < 1):
        $ 1321 "bajar≔pose_add(get_actual_tcp_pose(), bajada_broca)"
        global bajar= pose_add ( get_actual_tcp_pose (), bajada_broca)
        $ 1322 "bajar" "breakAfter"
        movel(bajar, a=0.004, v=0.004)
        $ 1323 "subir≔pose_sub(get_actual_tcp_pose(), bajada_broca)"
        global subir= pose_sub ( get_actual_tcp_pose (), bajada_broca)
        $ 1324 "Direction: Base Z+"
        global move_thread_flag_1324=0
        thread move_thread_1324():
          enter_critical
          move_thread_flag_1324 = 1
          local towardsPos=calculate_point_to_move_towards(p[0.0,0.0,0.0,0.0,0.0,0.0], [0.0,0.0,1.0], 0.002)
          movel(towardsPos, a=0.015, v=0.015)
          move_thread_flag_1324 = 2
          exit_critical
        end
        move_thread_flag_1324 = 0
        move_thread_han_1324 = run move_thread_1324()
        while (True):
          sleep(1.0E-10)
          if (move_thread_flag_1324 > 1):
            join move_thread_han_1324
            $ 1325 "Until (distance)"
            break
          end
          sync()
        end
        $ 1326 "Set CO[1]=Apagar"
        set_configurable_digital_out(1, False)
        $ 1327 "subir" "breakAfter"
        movel(subir, a=0.015, v=0.015)
        $ 1328 "bajada_broca≔pose_sub(bajada_broca, bajada)"
        global bajada_broca= pose_sub (bajada_broca, bajada)
        Loop_110 = Loop_110 + 1
      end
      $ 1329 "Direction: Base Z+"
      global move_thread_flag_1329=0
      thread move_thread_1329():
        enter_critical
        move_thread_flag_1329 = 1
        local towardsPos=calculate_point_to_move_towards(p[0.0,0.0,0.0,0.0,0.0,0.0], [0.0,0.0,1.0], 0.08)
        movel(towardsPos, a=0.15, v=0.1)
        move_thread_flag_1329 = 2
        exit_critical
      end
      move_thread_flag_1329 = 0
      move_thread_han_1329 = run move_thread_1329()
      while (True):
        sleep(1.0E-10)
        if (move_thread_flag_1329 > 1):
          join move_thread_han_1329
          $ 1330 "Until (distance)"
          break
        end
        sync()
      end
      $ 1331 "Set CO[1]=Apagar"
      set_configurable_digital_out(1, False)
      $ 1332 "barreno_actual≔barreno_actual+1"
      global barreno_actual=barreno_actual+1
      $ 1333 "Call Quitar_broca"
      Quitar_broca()
      $ 1334 "Call Poner_broca"
      Poner_broca()
    end
    $ 1335 "Popup: Linea8 con chica Terminada!"
    popup("Linea8 con chica Terminada!", "Mensaje", False, False, blocking=True)
    $ 1336 "Linea9"
    $ 1337 "Marcar_puntos"
    $ 1338 "MoveL"
    $ 1339 "Linea9_A" "breakAfter"
    movel(Linea9_A_p, a=0.5, v=0.1)
    $ 1340 "bajada_comprobacion"
    $ 1341 "Direction: Base Z-"
    global move_thread_flag_1341=0
    thread move_thread_1341():
      enter_critical
      move_thread_flag_1341 = 1
      local towardsPos=calculate_point_to_move_towards(p[0.0,0.0,0.0,0.0,0.0,0.0], [0.0,0.0,-1.0], 0.071)
      movel(towardsPos, a=0.15, v=0.1)
      move_thread_flag_1341 = 2
      exit_critical
    end
    move_thread_flag_1341 = 0
    move_thread_han_1341 = run move_thread_1341()
    while (True):
      sleep(1.0E-10)
      if (move_thread_flag_1341 > 1):
        join move_thread_han_1341
        $ 1342 "Until (distance)"
        break
      end
      sync()
    end
    $ 1343 "Direction: Base Z-"
    global move_thread_flag_1343=0
    thread move_thread_1343():
      enter_critical
      move_thread_flag_1343 = 1
      local towardsPos=calculate_point_to_move_towards(p[0.0,0.0,0.0,0.0,0.0,0.0], [0.0,0.0,-1.0], 1000.0)
      movel(towardsPos, a=0.007, v=0.007)
      move_thread_flag_1343 = 2
      exit_critical
    end
    move_thread_flag_1343 = 0
    move_thread_han_1343 = run move_thread_1343()
    while (True):
      local targetTcpDirection=get_target_tcp_speed()
      local stepsToRetract=tool_contact(direction=targetTcpDirection)
      if (stepsToRetract > 0):
        kill move_thread_han_1343
        stopl(0.02)
        local backTrackMovement=get_actual_joint_positions_history(stepsToRetract)
        local contactPose=get_forward_kin(backTrackMovement)
        local posDir=[targetTcpDirection[0],targetTcpDirection[1],targetTcpDirection[2]]
        local retractTo=contactPose
        if (norm(posDir) > 1e-6):
          local normalizedPosDir=normalize(posDir)
          local additionalRetraction=p[normalizedPosDir[0] * 0.0, normalizedPosDir[1] * 0.0, normalizedPosDir[2] * 0.0, 0, 0, 0]
          retractTo = pose_sub(contactPose, additionalRetraction)
        end
        movel(retractTo, a=0.02, v=0.1)
        $ 1344 "Until (tool_contact_detection)"
        break
      end
      sync()
    end
    $ 1345 "Direction: Base Z+"
    global move_thread_flag_1345=0
    thread move_thread_1345():
      enter_critical
      move_thread_flag_1345 = 1
      local towardsPos=calculate_point_to_move_towards(p[0.0,0.0,0.0,0.0,0.0,0.0], [0.0,0.0,1.0], 0.08)
      movel(towardsPos, a=0.15, v=0.1)
      move_thread_flag_1345 = 2
      exit_critical
    end
    move_thread_flag_1345 = 0
    move_thread_han_1345 = run move_thread_1345()
    while (True):
      sleep(1.0E-10)
      if (move_thread_flag_1345 > 1):
        join move_thread_han_1345
        $ 1346 "Until (distance)"
        break
      end
      sync()
    end
    $ 1347 "Linea9_B" "breakAfter"
    movel(Linea9_B_p, a=0.5, v=0.1)
    $ 1348 "bajada_comprobacion"
    $ 1349 "Direction: Base Z-"
    global move_thread_flag_1349=0
    thread move_thread_1349():
      enter_critical
      move_thread_flag_1349 = 1
      local towardsPos=calculate_point_to_move_towards(p[0.0,0.0,0.0,0.0,0.0,0.0], [0.0,0.0,-1.0], 0.071)
      movel(towardsPos, a=0.15, v=0.1)
      move_thread_flag_1349 = 2
      exit_critical
    end
    move_thread_flag_1349 = 0
    move_thread_han_1349 = run move_thread_1349()
    while (True):
      sleep(1.0E-10)
      if (move_thread_flag_1349 > 1):
        join move_thread_han_1349
        $ 1350 "Until (distance)"
        break
      end
      sync()
    end
    $ 1351 "Direction: Base Z-"
    global move_thread_flag_1351=0
    thread move_thread_1351():
      enter_critical
      move_thread_flag_1351 = 1
      local towardsPos=calculate_point_to_move_towards(p[0.0,0.0,0.0,0.0,0.0,0.0], [0.0,0.0,-1.0], 1000.0)
      movel(towardsPos, a=0.007, v=0.007)
      move_thread_flag_1351 = 2
      exit_critical
    end
    move_thread_flag_1351 = 0
    move_thread_han_1351 = run move_thread_1351()
    while (True):
      local targetTcpDirection=get_target_tcp_speed()
      local stepsToRetract=tool_contact(direction=targetTcpDirection)
      if (stepsToRetract > 0):
        kill move_thread_han_1351
        stopl(0.02)
        local backTrackMovement=get_actual_joint_positions_history(stepsToRetract)
        local contactPose=get_forward_kin(backTrackMovement)
        local posDir=[targetTcpDirection[0],targetTcpDirection[1],targetTcpDirection[2]]
        local retractTo=contactPose
        if (norm(posDir) > 1e-6):
          local normalizedPosDir=normalize(posDir)
          local additionalRetraction=p[normalizedPosDir[0] * 0.0, normalizedPosDir[1] * 0.0, normalizedPosDir[2] * 0.0, 0, 0, 0]
          retractTo = pose_sub(contactPose, additionalRetraction)
        end
        movel(retractTo, a=0.02, v=0.1)
        $ 1352 "Until (tool_contact_detection)"
        break
      end
      sync()
    end
    $ 1353 "Direction: Base Z+"
    global move_thread_flag_1353=0
    thread move_thread_1353():
      enter_critical
      move_thread_flag_1353 = 1
      local towardsPos=calculate_point_to_move_towards(p[0.0,0.0,0.0,0.0,0.0,0.0], [0.0,0.0,1.0], 0.08)
      movel(towardsPos, a=0.15, v=0.1)
      move_thread_flag_1353 = 2
      exit_critical
    end
    move_thread_flag_1353 = 0
    move_thread_han_1353 = run move_thread_1353()
    while (True):
      sleep(1.0E-10)
      if (move_thread_flag_1353 > 1):
        join move_thread_han_1353
        $ 1354 "Until (distance)"
        break
      end
      sync()
    end
    $ 1355 "AB"
    $ 1356 "'desbaste_inicial'"
    # 'desbaste_inicial'
    $ 1357 "bajada_broca≔p[0,0,-0.008,0,0,0]"
    global bajada_broca=p[0,0,-0.008,0,0,0]
    $ 1358 "barrenos_menos1≔2"
    global barrenos_menos1=2
    $ 1359 "barreno_actual≔0"
    global barreno_actual=0
    $ 1360 "Loop barreno_actual≤barrenos_menos1"
    while (barreno_actual <= barrenos_menos1):
      $ 1361 "Perforacion"
      $ 1362 "MoveL"
      $ 1363 "internos≔interpolate_pose(Linea9_A, Linea9_B, barreno_actual/barrenos_menos1)"
      global internos= interpolate_pose (Linea9_A_p, Linea9_B_p, barreno_actual/barrenos_menos1)
      $ 1364 "internos" "breakAfter"
      movel(internos, a=0.5, v=0.1)
      $ 1365 "'desbaste_inicial'"
      # 'desbaste_inicial'
      $ 1366 "bajada_broca≔p[0,0,-0.024,0,0,0]"
      global bajada_broca=p[0,0,-0.024,0,0,0]
      $ 1367 "bajada≔p[0,0,0.024,0,0,0]"
      global bajada=p[0,0,0.024,0,0,0]
      $ 1368 "Direction: Base Z-"
      global move_thread_flag_1368=0
      thread move_thread_1368():
        enter_critical
        move_thread_flag_1368 = 1
        local towardsPos=calculate_point_to_move_towards(p[0.0,0.0,0.0,0.0,0.0,0.0], [0.0,0.0,-1.0], 0.071)
        movel(towardsPos, a=0.15, v=0.1)
        move_thread_flag_1368 = 2
        exit_critical
      end
      move_thread_flag_1368 = 0
      move_thread_han_1368 = run move_thread_1368()
      while (True):
        sleep(1.0E-10)
        if (move_thread_flag_1368 > 1):
          join move_thread_han_1368
          $ 1369 "Until (distance)"
          break
        end
        sync()
      end
      $ 1370 "Direction: Base Z-"
      global move_thread_flag_1370=0
      thread move_thread_1370():
        enter_critical
        move_thread_flag_1370 = 1
        local towardsPos=calculate_point_to_move_towards(p[0.0,0.0,0.0,0.0,0.0,0.0], [0.0,0.0,-1.0], 1000.0)
        movel(towardsPos, a=0.007, v=0.007)
        move_thread_flag_1370 = 2
        exit_critical
      end
      move_thread_flag_1370 = 0
      move_thread_han_1370 = run move_thread_1370()
      while (True):
        local targetTcpDirection=get_target_tcp_speed()
        local stepsToRetract=tool_contact(direction=targetTcpDirection)
        if (stepsToRetract > 0):
          kill move_thread_han_1370
          stopl(0.02)
          local backTrackMovement=get_actual_joint_positions_history(stepsToRetract)
          local contactPose=get_forward_kin(backTrackMovement)
          local posDir=[targetTcpDirection[0],targetTcpDirection[1],targetTcpDirection[2]]
          local retractTo=contactPose
          if (norm(posDir) > 1e-6):
            local normalizedPosDir=normalize(posDir)
            local additionalRetraction=p[normalizedPosDir[0] * 0.0, normalizedPosDir[1] * 0.0, normalizedPosDir[2] * 0.0, 0, 0, 0]
            retractTo = pose_sub(contactPose, additionalRetraction)
          end
          movel(retractTo, a=0.02, v=0.1)
          $ 1371 "Until (tool_contact_detection)"
          break
        end
        sync()
      end
      $ 1372 "Popup: punto contacto alanzdo"
      popup("punto contacto alanzdo", "Mensaje", False, False, blocking=True)
      $ 1373 "Direction: Base Z+"
      global move_thread_flag_1373=0
      thread move_thread_1373():
        enter_critical
        move_thread_flag_1373 = 1
        local towardsPos=calculate_point_to_move_towards(p[0.0,0.0,0.0,0.0,0.0,0.0], [0.0,0.0,1.0], 0.007)
        movel(towardsPos, a=0.015, v=0.015)
        move_thread_flag_1373 = 2
        exit_critical
      end
      move_thread_flag_1373 = 0
      move_thread_han_1373 = run move_thread_1373()
      while (True):
        sleep(1.0E-10)
        if (move_thread_flag_1373 > 1):
          join move_thread_han_1373
          $ 1374 "Until (distance)"
          break
        end
        sync()
      end
      $ 1375 "Wait: 0.3"
      sleep(0.3)
      $ 1376 "Set CO[1]=Encender"
      set_configurable_digital_out(1, True)
      $ 1377 "Wait: 0.3"
      sleep(0.3)
      $ 1378 "Loop 1 times"
      Loop_114 = 0
      while (Loop_114 < 1):
        $ 1379 "bajar≔pose_add(get_actual_tcp_pose(), bajada_broca)"
        global bajar= pose_add ( get_actual_tcp_pose (), bajada_broca)
        $ 1380 "bajar" "breakAfter"
        movel(bajar, a=0.004, v=0.004)
        $ 1381 "subir≔pose_sub(get_actual_tcp_pose(), bajada_broca)"
        global subir= pose_sub ( get_actual_tcp_pose (), bajada_broca)
        $ 1382 "Direction: Base Z+"
        global move_thread_flag_1382=0
        thread move_thread_1382():
          enter_critical
          move_thread_flag_1382 = 1
          local towardsPos=calculate_point_to_move_towards(p[0.0,0.0,0.0,0.0,0.0,0.0], [0.0,0.0,1.0], 0.002)
          movel(towardsPos, a=0.015, v=0.015)
          move_thread_flag_1382 = 2
          exit_critical
        end
        move_thread_flag_1382 = 0
        move_thread_han_1382 = run move_thread_1382()
        while (True):
          sleep(1.0E-10)
          if (move_thread_flag_1382 > 1):
            join move_thread_han_1382
            $ 1383 "Until (distance)"
            break
          end
          sync()
        end
        $ 1384 "Set CO[1]=Apagar"
        set_configurable_digital_out(1, False)
        $ 1385 "subir" "breakAfter"
        movel(subir, a=0.015, v=0.015)
        $ 1386 "bajada_broca≔pose_sub(bajada_broca, bajada)"
        global bajada_broca= pose_sub (bajada_broca, bajada)
        Loop_114 = Loop_114 + 1
      end
      $ 1387 "Direction: Base Z+"
      global move_thread_flag_1387=0
      thread move_thread_1387():
        enter_critical
        move_thread_flag_1387 = 1
        local towardsPos=calculate_point_to_move_towards(p[0.0,0.0,0.0,0.0,0.0,0.0], [0.0,0.0,1.0], 0.08)
        movel(towardsPos, a=0.15, v=0.1)
        move_thread_flag_1387 = 2
        exit_critical
      end
      move_thread_flag_1387 = 0
      move_thread_han_1387 = run move_thread_1387()
      while (True):
        sleep(1.0E-10)
        if (move_thread_flag_1387 > 1):
          join move_thread_han_1387
          $ 1388 "Until (distance)"
          break
        end
        sync()
      end
      $ 1389 "Set CO[1]=Apagar"
      set_configurable_digital_out(1, False)
      $ 1390 "barreno_actual≔barreno_actual+1"
      global barreno_actual=barreno_actual+1
      $ 1391 "Call Quitar_broca"
      Quitar_broca()
      $ 1392 "Call Poner_broca"
      Poner_broca()
    end
    $ 1393 "Popup: Linea9 con chica Terminada!"
    popup("Linea9 con chica Terminada!", "Mensaje", False, False, blocking=True)
    $ 1394 "Linea10"
    $ 1395 "Marcar_puntos"
    $ 1396 "MoveL"
    $ 1397 "Home2" "breakAfter"
    movel(Home2_p, a=0.5, v=0.1)
    $ 1398 "Linea10_A" "breakAfter"
    movel(Linea10_A_p, a=0.5, v=0.1)
    $ 1399 "bajada_comprobacion"
    $ 1400 "Direction: Base Z-"
    global move_thread_flag_1400=0
    thread move_thread_1400():
      enter_critical
      move_thread_flag_1400 = 1
      local towardsPos=calculate_point_to_move_towards(p[0.0,0.0,0.0,0.0,0.0,0.0], [0.0,0.0,-1.0], 0.071)
      movel(towardsPos, a=0.15, v=0.1)
      move_thread_flag_1400 = 2
      exit_critical
    end
    move_thread_flag_1400 = 0
    move_thread_han_1400 = run move_thread_1400()
    while (True):
      sleep(1.0E-10)
      if (move_thread_flag_1400 > 1):
        join move_thread_han_1400
        $ 1401 "Until (distance)"
        break
      end
      sync()
    end
    $ 1402 "Direction: Base Z-"
    global move_thread_flag_1402=0
    thread move_thread_1402():
      enter_critical
      move_thread_flag_1402 = 1
      local towardsPos=calculate_point_to_move_towards(p[0.0,0.0,0.0,0.0,0.0,0.0], [0.0,0.0,-1.0], 1000.0)
      movel(towardsPos, a=0.007, v=0.007)
      move_thread_flag_1402 = 2
      exit_critical
    end
    move_thread_flag_1402 = 0
    move_thread_han_1402 = run move_thread_1402()
    while (True):
      local targetTcpDirection=get_target_tcp_speed()
      local stepsToRetract=tool_contact(direction=targetTcpDirection)
      if (stepsToRetract > 0):
        kill move_thread_han_1402
        stopl(0.02)
        local backTrackMovement=get_actual_joint_positions_history(stepsToRetract)
        local contactPose=get_forward_kin(backTrackMovement)
        local posDir=[targetTcpDirection[0],targetTcpDirection[1],targetTcpDirection[2]]
        local retractTo=contactPose
        if (norm(posDir) > 1e-6):
          local normalizedPosDir=normalize(posDir)
          local additionalRetraction=p[normalizedPosDir[0] * 0.0, normalizedPosDir[1] * 0.0, normalizedPosDir[2] * 0.0, 0, 0, 0]
          retractTo = pose_sub(contactPose, additionalRetraction)
        end
        movel(retractTo, a=0.02, v=0.1)
        $ 1403 "Until (tool_contact_detection)"
        break
      end
      sync()
    end
    $ 1404 "Direction: Base Z+"
    global move_thread_flag_1404=0
    thread move_thread_1404():
      enter_critical
      move_thread_flag_1404 = 1
      local towardsPos=calculate_point_to_move_towards(p[0.0,0.0,0.0,0.0,0.0,0.0], [0.0,0.0,1.0], 0.08)
      movel(towardsPos, a=0.15, v=0.1)
      move_thread_flag_1404 = 2
      exit_critical
    end
    move_thread_flag_1404 = 0
    move_thread_han_1404 = run move_thread_1404()
    while (True):
      sleep(1.0E-10)
      if (move_thread_flag_1404 > 1):
        join move_thread_han_1404
        $ 1405 "Until (distance)"
        break
      end
      sync()
    end
    $ 1406 "Linea10_B" "breakAfter"
    movel(Linea10_B_p, a=0.5, v=0.1)
    $ 1407 "bajada_comprobacion"
    $ 1408 "Direction: Base Z-"
    global move_thread_flag_1408=0
    thread move_thread_1408():
      enter_critical
      move_thread_flag_1408 = 1
      local towardsPos=calculate_point_to_move_towards(p[0.0,0.0,0.0,0.0,0.0,0.0], [0.0,0.0,-1.0], 0.071)
      movel(towardsPos, a=0.15, v=0.1)
      move_thread_flag_1408 = 2
      exit_critical
    end
    move_thread_flag_1408 = 0
    move_thread_han_1408 = run move_thread_1408()
    while (True):
      sleep(1.0E-10)
      if (move_thread_flag_1408 > 1):
        join move_thread_han_1408
        $ 1409 "Until (distance)"
        break
      end
      sync()
    end
    $ 1410 "Direction: Base Z-"
    global move_thread_flag_1410=0
    thread move_thread_1410():
      enter_critical
      move_thread_flag_1410 = 1
      local towardsPos=calculate_point_to_move_towards(p[0.0,0.0,0.0,0.0,0.0,0.0], [0.0,0.0,-1.0], 1000.0)
      movel(towardsPos, a=0.007, v=0.007)
      move_thread_flag_1410 = 2
      exit_critical
    end
    move_thread_flag_1410 = 0
    move_thread_han_1410 = run move_thread_1410()
    while (True):
      local targetTcpDirection=get_target_tcp_speed()
      local stepsToRetract=tool_contact(direction=targetTcpDirection)
      if (stepsToRetract > 0):
        kill move_thread_han_1410
        stopl(0.02)
        local backTrackMovement=get_actual_joint_positions_history(stepsToRetract)
        local contactPose=get_forward_kin(backTrackMovement)
        local posDir=[targetTcpDirection[0],targetTcpDirection[1],targetTcpDirection[2]]
        local retractTo=contactPose
        if (norm(posDir) > 1e-6):
          local normalizedPosDir=normalize(posDir)
          local additionalRetraction=p[normalizedPosDir[0] * 0.0, normalizedPosDir[1] * 0.0, normalizedPosDir[2] * 0.0, 0, 0, 0]
          retractTo = pose_sub(contactPose, additionalRetraction)
        end
        movel(retractTo, a=0.02, v=0.1)
        $ 1411 "Until (tool_contact_detection)"
        break
      end
      sync()
    end
    $ 1412 "Direction: Base Z+"
    global move_thread_flag_1412=0
    thread move_thread_1412():
      enter_critical
      move_thread_flag_1412 = 1
      local towardsPos=calculate_point_to_move_towards(p[0.0,0.0,0.0,0.0,0.0,0.0], [0.0,0.0,1.0], 0.08)
      movel(towardsPos, a=0.15, v=0.1)
      move_thread_flag_1412 = 2
      exit_critical
    end
    move_thread_flag_1412 = 0
    move_thread_han_1412 = run move_thread_1412()
    while (True):
      sleep(1.0E-10)
      if (move_thread_flag_1412 > 1):
        join move_thread_han_1412
        $ 1413 "Until (distance)"
        break
      end
      sync()
    end
    $ 1414 "AB"
    $ 1415 "'desbaste_inicial'"
    # 'desbaste_inicial'
    $ 1416 "bajada_broca≔p[0,0,-0.008,0,0,0]"
    global bajada_broca=p[0,0,-0.008,0,0,0]
    $ 1417 "barrenos_menos1≔2"
    global barrenos_menos1=2
    $ 1418 "barreno_actual≔0"
    global barreno_actual=0
    $ 1419 "Loop barreno_actual≤barrenos_menos1"
    while (barreno_actual <= barrenos_menos1):
      $ 1420 "Perforacion"
      $ 1421 "MoveL"
      $ 1422 "internos≔interpolate_pose(Linea10_A, Linea10_B, barreno_actual/barrenos_menos1)"
      global internos= interpolate_pose (Linea10_A_p, Linea10_B_p, barreno_actual/barrenos_menos1)
      $ 1423 "internos" "breakAfter"
      movel(internos, a=0.5, v=0.1)
      $ 1424 "'desbaste_inicial'"
      # 'desbaste_inicial'
      $ 1425 "bajada_broca≔p[0,0,-0.024,0,0,0]"
      global bajada_broca=p[0,0,-0.024,0,0,0]
      $ 1426 "bajada≔p[0,0,0.024,0,0,0]"
      global bajada=p[0,0,0.024,0,0,0]
      $ 1427 "Direction: Base Z-"
      global move_thread_flag_1427=0
      thread move_thread_1427():
        enter_critical
        move_thread_flag_1427 = 1
        local towardsPos=calculate_point_to_move_towards(p[0.0,0.0,0.0,0.0,0.0,0.0], [0.0,0.0,-1.0], 0.071)
        movel(towardsPos, a=0.15, v=0.1)
        move_thread_flag_1427 = 2
        exit_critical
      end
      move_thread_flag_1427 = 0
      move_thread_han_1427 = run move_thread_1427()
      while (True):
        sleep(1.0E-10)
        if (move_thread_flag_1427 > 1):
          join move_thread_han_1427
          $ 1428 "Until (distance)"
          break
        end
        sync()
      end
      $ 1429 "Direction: Base Z-"
      global move_thread_flag_1429=0
      thread move_thread_1429():
        enter_critical
        move_thread_flag_1429 = 1
        local towardsPos=calculate_point_to_move_towards(p[0.0,0.0,0.0,0.0,0.0,0.0], [0.0,0.0,-1.0], 1000.0)
        movel(towardsPos, a=0.007, v=0.007)
        move_thread_flag_1429 = 2
        exit_critical
      end
      move_thread_flag_1429 = 0
      move_thread_han_1429 = run move_thread_1429()
      while (True):
        local targetTcpDirection=get_target_tcp_speed()
        local stepsToRetract=tool_contact(direction=targetTcpDirection)
        if (stepsToRetract > 0):
          kill move_thread_han_1429
          stopl(0.02)
          local backTrackMovement=get_actual_joint_positions_history(stepsToRetract)
          local contactPose=get_forward_kin(backTrackMovement)
          local posDir=[targetTcpDirection[0],targetTcpDirection[1],targetTcpDirection[2]]
          local retractTo=contactPose
          if (norm(posDir) > 1e-6):
            local normalizedPosDir=normalize(posDir)
            local additionalRetraction=p[normalizedPosDir[0] * 0.0, normalizedPosDir[1] * 0.0, normalizedPosDir[2] * 0.0, 0, 0, 0]
            retractTo = pose_sub(contactPose, additionalRetraction)
          end
          movel(retractTo, a=0.02, v=0.1)
          $ 1430 "Until (tool_contact_detection)"
          break
        end
        sync()
      end
      $ 1431 "Popup: punto contacto alanzdo"
      popup("punto contacto alanzdo", "Mensaje", False, False, blocking=True)
      $ 1432 "Direction: Base Z+"
      global move_thread_flag_1432=0
      thread move_thread_1432():
        enter_critical
        move_thread_flag_1432 = 1
        local towardsPos=calculate_point_to_move_towards(p[0.0,0.0,0.0,0.0,0.0,0.0], [0.0,0.0,1.0], 0.007)
        movel(towardsPos, a=0.015, v=0.015)
        move_thread_flag_1432 = 2
        exit_critical
      end
      move_thread_flag_1432 = 0
      move_thread_han_1432 = run move_thread_1432()
      while (True):
        sleep(1.0E-10)
        if (move_thread_flag_1432 > 1):
          join move_thread_han_1432
          $ 1433 "Until (distance)"
          break
        end
        sync()
      end
      $ 1434 "Wait: 0.3"
      sleep(0.3)
      $ 1435 "Set CO[1]=Encender"
      set_configurable_digital_out(1, True)
      $ 1436 "Wait: 0.3"
      sleep(0.3)
      $ 1437 "Loop 1 times"
      Loop_118 = 0
      while (Loop_118 < 1):
        $ 1438 "bajar≔pose_add(get_actual_tcp_pose(), bajada_broca)"
        global bajar= pose_add ( get_actual_tcp_pose (), bajada_broca)
        $ 1439 "bajar" "breakAfter"
        movel(bajar, a=0.004, v=0.004)
        $ 1440 "subir≔pose_sub(get_actual_tcp_pose(), bajada_broca)"
        global subir= pose_sub ( get_actual_tcp_pose (), bajada_broca)
        $ 1441 "Direction: Base Z+"
        global move_thread_flag_1441=0
        thread move_thread_1441():
          enter_critical
          move_thread_flag_1441 = 1
          local towardsPos=calculate_point_to_move_towards(p[0.0,0.0,0.0,0.0,0.0,0.0], [0.0,0.0,1.0], 0.002)
          movel(towardsPos, a=0.015, v=0.015)
          move_thread_flag_1441 = 2
          exit_critical
        end
        move_thread_flag_1441 = 0
        move_thread_han_1441 = run move_thread_1441()
        while (True):
          sleep(1.0E-10)
          if (move_thread_flag_1441 > 1):
            join move_thread_han_1441
            $ 1442 "Until (distance)"
            break
          end
          sync()
        end
        $ 1443 "Set CO[1]=Apagar"
        set_configurable_digital_out(1, False)
        $ 1444 "subir" "breakAfter"
        movel(subir, a=0.015, v=0.015)
        $ 1445 "bajada_broca≔pose_sub(bajada_broca, bajada)"
        global bajada_broca= pose_sub (bajada_broca, bajada)
        Loop_118 = Loop_118 + 1
      end
      $ 1446 "Direction: Base Z+"
      global move_thread_flag_1446=0
      thread move_thread_1446():
        enter_critical
        move_thread_flag_1446 = 1
        local towardsPos=calculate_point_to_move_towards(p[0.0,0.0,0.0,0.0,0.0,0.0], [0.0,0.0,1.0], 0.08)
        movel(towardsPos, a=0.15, v=0.1)
        move_thread_flag_1446 = 2
        exit_critical
      end
      move_thread_flag_1446 = 0
      move_thread_han_1446 = run move_thread_1446()
      while (True):
        sleep(1.0E-10)
        if (move_thread_flag_1446 > 1):
          join move_thread_han_1446
          $ 1447 "Until (distance)"
          break
        end
        sync()
      end
      $ 1448 "Set CO[1]=Apagar"
      set_configurable_digital_out(1, False)
      $ 1449 "barreno_actual≔barreno_actual+1"
      global barreno_actual=barreno_actual+1
    end
    $ 1452 "Popup: Linea10 con chica Terminada!"
    popup("Linea10 con chica Terminada!", "Mensaje", False, False, blocking=True)
    $ 1453 "Linea11"
    $ 1454 "Marcar_puntos"
    $ 1455 "MoveL"
    $ 1456 "Linea11_A" "breakAfter"
    movel(Linea11_A_p, a=0.5, v=0.1)
    $ 1457 "bajada_comprobacion"
    $ 1458 "Direction: Base Z-"
    global move_thread_flag_1458=0
    thread move_thread_1458():
      enter_critical
      move_thread_flag_1458 = 1
      local towardsPos=calculate_point_to_move_towards(p[0.0,0.0,0.0,0.0,0.0,0.0], [0.0,0.0,-1.0], 0.071)
      movel(towardsPos, a=0.15, v=0.1)
      move_thread_flag_1458 = 2
      exit_critical
    end
    move_thread_flag_1458 = 0
    move_thread_han_1458 = run move_thread_1458()
    while (True):
      sleep(1.0E-10)
      if (move_thread_flag_1458 > 1):
        join move_thread_han_1458
        $ 1459 "Until (distance)"
        break
      end
      sync()
    end
    $ 1460 "Direction: Base Z-"
    global move_thread_flag_1460=0
    thread move_thread_1460():
      enter_critical
      move_thread_flag_1460 = 1
      local towardsPos=calculate_point_to_move_towards(p[0.0,0.0,0.0,0.0,0.0,0.0], [0.0,0.0,-1.0], 1000.0)
      movel(towardsPos, a=0.007, v=0.007)
      move_thread_flag_1460 = 2
      exit_critical
    end
    move_thread_flag_1460 = 0
    move_thread_han_1460 = run move_thread_1460()
    while (True):
      local targetTcpDirection=get_target_tcp_speed()
      local stepsToRetract=tool_contact(direction=targetTcpDirection)
      if (stepsToRetract > 0):
        kill move_thread_han_1460
        stopl(0.02)
        local backTrackMovement=get_actual_joint_positions_history(stepsToRetract)
        local contactPose=get_forward_kin(backTrackMovement)
        local posDir=[targetTcpDirection[0],targetTcpDirection[1],targetTcpDirection[2]]
        local retractTo=contactPose
        if (norm(posDir) > 1e-6):
          local normalizedPosDir=normalize(posDir)
          local additionalRetraction=p[normalizedPosDir[0] * 0.0, normalizedPosDir[1] * 0.0, normalizedPosDir[2] * 0.0, 0, 0, 0]
          retractTo = pose_sub(contactPose, additionalRetraction)
        end
        movel(retractTo, a=0.02, v=0.1)
        $ 1461 "Until (tool_contact_detection)"
        break
      end
      sync()
    end
    $ 1462 "Direction: Base Z+"
    global move_thread_flag_1462=0
    thread move_thread_1462():
      enter_critical
      move_thread_flag_1462 = 1
      local towardsPos=calculate_point_to_move_towards(p[0.0,0.0,0.0,0.0,0.0,0.0], [0.0,0.0,1.0], 0.08)
      movel(towardsPos, a=0.15, v=0.1)
      move_thread_flag_1462 = 2
      exit_critical
    end
    move_thread_flag_1462 = 0
    move_thread_han_1462 = run move_thread_1462()
    while (True):
      sleep(1.0E-10)
      if (move_thread_flag_1462 > 1):
        join move_thread_han_1462
        $ 1463 "Until (distance)"
        break
      end
      sync()
    end
    $ 1464 "Linea11_B" "breakAfter"
    movel(Linea11_B_p, a=0.5, v=0.1)
    $ 1465 "bajada_comprobacion"
    $ 1466 "Direction: Base Z-"
    global move_thread_flag_1466=0
    thread move_thread_1466():
      enter_critical
      move_thread_flag_1466 = 1
      local towardsPos=calculate_point_to_move_towards(p[0.0,0.0,0.0,0.0,0.0,0.0], [0.0,0.0,-1.0], 0.071)
      movel(towardsPos, a=0.15, v=0.1)
      move_thread_flag_1466 = 2
      exit_critical
    end
    move_thread_flag_1466 = 0
    move_thread_han_1466 = run move_thread_1466()
    while (True):
      sleep(1.0E-10)
      if (move_thread_flag_1466 > 1):
        join move_thread_han_1466
        $ 1467 "Until (distance)"
        break
      end
      sync()
    end
    $ 1468 "Direction: Base Z-"
    global move_thread_flag_1468=0
    thread move_thread_1468():
      enter_critical
      move_thread_flag_1468 = 1
      local towardsPos=calculate_point_to_move_towards(p[0.0,0.0,0.0,0.0,0.0,0.0], [0.0,0.0,-1.0], 1000.0)
      movel(towardsPos, a=0.007, v=0.007)
      move_thread_flag_1468 = 2
      exit_critical
    end
    move_thread_flag_1468 = 0
    move_thread_han_1468 = run move_thread_1468()
    while (True):
      local targetTcpDirection=get_target_tcp_speed()
      local stepsToRetract=tool_contact(direction=targetTcpDirection)
      if (stepsToRetract > 0):
        kill move_thread_han_1468
        stopl(0.02)
        local backTrackMovement=get_actual_joint_positions_history(stepsToRetract)
        local contactPose=get_forward_kin(backTrackMovement)
        local posDir=[targetTcpDirection[0],targetTcpDirection[1],targetTcpDirection[2]]
        local retractTo=contactPose
        if (norm(posDir) > 1e-6):
          local normalizedPosDir=normalize(posDir)
          local additionalRetraction=p[normalizedPosDir[0] * 0.0, normalizedPosDir[1] * 0.0, normalizedPosDir[2] * 0.0, 0, 0, 0]
          retractTo = pose_sub(contactPose, additionalRetraction)
        end
        movel(retractTo, a=0.02, v=0.1)
        $ 1469 "Until (tool_contact_detection)"
        break
      end
      sync()
    end
    $ 1470 "Direction: Base Z+"
    global move_thread_flag_1470=0
    thread move_thread_1470():
      enter_critical
      move_thread_flag_1470 = 1
      local towardsPos=calculate_point_to_move_towards(p[0.0,0.0,0.0,0.0,0.0,0.0], [0.0,0.0,1.0], 0.08)
      movel(towardsPos, a=0.15, v=0.1)
      move_thread_flag_1470 = 2
      exit_critical
    end
    move_thread_flag_1470 = 0
    move_thread_han_1470 = run move_thread_1470()
    while (True):
      sleep(1.0E-10)
      if (move_thread_flag_1470 > 1):
        join move_thread_han_1470
        $ 1471 "Until (distance)"
        break
      end
      sync()
    end
    $ 1472 "AB"
    $ 1473 "'desbaste_inicial'"
    # 'desbaste_inicial'
    $ 1474 "bajada_broca≔p[0,0,-0.008,0,0,0]"
    global bajada_broca=p[0,0,-0.008,0,0,0]
    $ 1475 "barrenos_menos1≔2"
    global barrenos_menos1=2
    $ 1476 "barreno_actual≔0"
    global barreno_actual=0
    $ 1477 "Loop barreno_actual≤barrenos_menos1"
    while (barreno_actual <= barrenos_menos1):
      $ 1478 "Perforacion"
      $ 1479 "MoveL"
      $ 1482 "internos≔interpolate_pose(Linea11_A, Linea11_B, barreno_actual/barrenos_menos1)"
      global internos= interpolate_pose (Linea11_A_p, Linea11_B_p, barreno_actual/barrenos_menos1)
      $ 1483 "internos" "breakAfter"
      movel(internos, a=0.5, v=0.1)
      $ 1484 "'desbaste_inicial'"
      # 'desbaste_inicial'
      $ 1485 "bajada_broca≔p[0,0,-0.024,0,0,0]"
      global bajada_broca=p[0,0,-0.024,0,0,0]
      $ 1486 "bajada≔p[0,0,0.024,0,0,0]"
      global bajada=p[0,0,0.024,0,0,0]
      $ 1487 "Direction: Base Z-"
      global move_thread_flag_1487=0
      thread move_thread_1487():
        enter_critical
        move_thread_flag_1487 = 1
        local towardsPos=calculate_point_to_move_towards(p[0.0,0.0,0.0,0.0,0.0,0.0], [0.0,0.0,-1.0], 0.071)
        movel(towardsPos, a=0.15, v=0.1)
        move_thread_flag_1487 = 2
        exit_critical
      end
      move_thread_flag_1487 = 0
      move_thread_han_1487 = run move_thread_1487()
      while (True):
        sleep(1.0E-10)
        if (move_thread_flag_1487 > 1):
          join move_thread_han_1487
          $ 1488 "Until (distance)"
          break
        end
        sync()
      end
      $ 1489 "Direction: Base Z-"
      global move_thread_flag_1489=0
      thread move_thread_1489():
        enter_critical
        move_thread_flag_1489 = 1
        local towardsPos=calculate_point_to_move_towards(p[0.0,0.0,0.0,0.0,0.0,0.0], [0.0,0.0,-1.0], 1000.0)
        movel(towardsPos, a=0.007, v=0.007)
        move_thread_flag_1489 = 2
        exit_critical
      end
      move_thread_flag_1489 = 0
      move_thread_han_1489 = run move_thread_1489()
      while (True):
        local targetTcpDirection=get_target_tcp_speed()
        local stepsToRetract=tool_contact(direction=targetTcpDirection)
        if (stepsToRetract > 0):
          kill move_thread_han_1489
          stopl(0.02)
          local backTrackMovement=get_actual_joint_positions_history(stepsToRetract)
          local contactPose=get_forward_kin(backTrackMovement)
          local posDir=[targetTcpDirection[0],targetTcpDirection[1],targetTcpDirection[2]]
          local retractTo=contactPose
          if (norm(posDir) > 1e-6):
            local normalizedPosDir=normalize(posDir)
            local additionalRetraction=p[normalizedPosDir[0] * 0.0, normalizedPosDir[1] * 0.0, normalizedPosDir[2] * 0.0, 0, 0, 0]
            retractTo = pose_sub(contactPose, additionalRetraction)
          end
          movel(retractTo, a=0.02, v=0.1)
          $ 1490 "Until (tool_contact_detection)"
          break
        end
        sync()
      end
      $ 1491 "Popup: punto contacto alanzdo"
      popup("punto contacto alanzdo", "Mensaje", False, False, blocking=True)
      $ 1492 "Direction: Base Z+"
      global move_thread_flag_1492=0
      thread move_thread_1492():
        enter_critical
        move_thread_flag_1492 = 1
        local towardsPos=calculate_point_to_move_towards(p[0.0,0.0,0.0,0.0,0.0,0.0], [0.0,0.0,1.0], 0.007)
        movel(towardsPos, a=0.015, v=0.015)
        move_thread_flag_1492 = 2
        exit_critical
      end
      move_thread_flag_1492 = 0
      move_thread_han_1492 = run move_thread_1492()
      while (True):
        sleep(1.0E-10)
        if (move_thread_flag_1492 > 1):
          join move_thread_han_1492
          $ 1493 "Until (distance)"
          break
        end
        sync()
      end
      $ 1494 "Wait: 0.3"
      sleep(0.3)
      $ 1495 "Set CO[1]=Encender"
      set_configurable_digital_out(1, True)
      $ 1496 "Wait: 0.3"
      sleep(0.3)
      $ 1497 "Loop 1 times"
      Loop_122 = 0
      while (Loop_122 < 1):
        $ 1498 "bajar≔pose_add(get_actual_tcp_pose(), bajada_broca)"
        global bajar= pose_add ( get_actual_tcp_pose (), bajada_broca)
        $ 1499 "bajar" "breakAfter"
        movel(bajar, a=0.004, v=0.004)
        $ 1500 "subir≔pose_sub(get_actual_tcp_pose(), bajada_broca)"
        global subir= pose_sub ( get_actual_tcp_pose (), bajada_broca)
        $ 1501 "Direction: Base Z+"
        global move_thread_flag_1501=0
        thread move_thread_1501():
          enter_critical
          move_thread_flag_1501 = 1
          local towardsPos=calculate_point_to_move_towards(p[0.0,0.0,0.0,0.0,0.0,0.0], [0.0,0.0,1.0], 0.002)
          movel(towardsPos, a=0.015, v=0.015)
          move_thread_flag_1501 = 2
          exit_critical
        end
        move_thread_flag_1501 = 0
        move_thread_han_1501 = run move_thread_1501()
        while (True):
          sleep(1.0E-10)
          if (move_thread_flag_1501 > 1):
            join move_thread_han_1501
            $ 1502 "Until (distance)"
            break
          end
          sync()
        end
        $ 1503 "Set CO[1]=Apagar"
        set_configurable_digital_out(1, False)
        $ 1504 "subir" "breakAfter"
        movel(subir, a=0.015, v=0.015)
        $ 1505 "bajada_broca≔pose_sub(bajada_broca, bajada)"
        global bajada_broca= pose_sub (bajada_broca, bajada)
        Loop_122 = Loop_122 + 1
      end
      $ 1506 "Direction: Base Z+"
      global move_thread_flag_1506=0
      thread move_thread_1506():
        enter_critical
        move_thread_flag_1506 = 1
        local towardsPos=calculate_point_to_move_towards(p[0.0,0.0,0.0,0.0,0.0,0.0], [0.0,0.0,1.0], 0.08)
        movel(towardsPos, a=0.15, v=0.1)
        move_thread_flag_1506 = 2
        exit_critical
      end
      move_thread_flag_1506 = 0
      move_thread_han_1506 = run move_thread_1506()
      while (True):
        sleep(1.0E-10)
        if (move_thread_flag_1506 > 1):
          join move_thread_han_1506
          $ 1507 "Until (distance)"
          break
        end
        sync()
      end
      $ 1508 "Set CO[1]=Apagar"
      set_configurable_digital_out(1, False)
      $ 1509 "barreno_actual≔barreno_actual+1"
      global barreno_actual=barreno_actual+1
    end
    $ 1512 "Popup: Linea11 con chica Terminada!"
    popup("Linea11 con chica Terminada!", "Mensaje", False, False, blocking=True)
    $ 1513 "Linea12"
    $ 1514 "Marcar_puntos"
    $ 1515 "MoveL"
    $ 1516 "Linea12_A" "breakAfter"
    movel(Linea12_A_p, a=0.5, v=0.1)
    $ 1517 "bajada_comprobacion"
    $ 1518 "Direction: Base Z-"
    global move_thread_flag_1518=0
    thread move_thread_1518():
      enter_critical
      move_thread_flag_1518 = 1
      local towardsPos=calculate_point_to_move_towards(p[0.0,0.0,0.0,0.0,0.0,0.0], [0.0,0.0,-1.0], 0.071)
      movel(towardsPos, a=0.15, v=0.1)
      move_thread_flag_1518 = 2
      exit_critical
    end
    move_thread_flag_1518 = 0
    move_thread_han_1518 = run move_thread_1518()
    while (True):
      sleep(1.0E-10)
      if (move_thread_flag_1518 > 1):
        join move_thread_han_1518
        $ 1519 "Until (distance)"
        break
      end
      sync()
    end
    $ 1520 "Direction: Base Z-"
    global move_thread_flag_1520=0
    thread move_thread_1520():
      enter_critical
      move_thread_flag_1520 = 1
      local towardsPos=calculate_point_to_move_towards(p[0.0,0.0,0.0,0.0,0.0,0.0], [0.0,0.0,-1.0], 1000.0)
      movel(towardsPos, a=0.007, v=0.007)
      move_thread_flag_1520 = 2
      exit_critical
    end
    move_thread_flag_1520 = 0
    move_thread_han_1520 = run move_thread_1520()
    while (True):
      local targetTcpDirection=get_target_tcp_speed()
      local stepsToRetract=tool_contact(direction=targetTcpDirection)
      if (stepsToRetract > 0):
        kill move_thread_han_1520
        stopl(0.02)
        local backTrackMovement=get_actual_joint_positions_history(stepsToRetract)
        local contactPose=get_forward_kin(backTrackMovement)
        local posDir=[targetTcpDirection[0],targetTcpDirection[1],targetTcpDirection[2]]
        local retractTo=contactPose
        if (norm(posDir) > 1e-6):
          local normalizedPosDir=normalize(posDir)
          local additionalRetraction=p[normalizedPosDir[0] * 0.0, normalizedPosDir[1] * 0.0, normalizedPosDir[2] * 0.0, 0, 0, 0]
          retractTo = pose_sub(contactPose, additionalRetraction)
        end
        movel(retractTo, a=0.02, v=0.1)
        $ 1521 "Until (tool_contact_detection)"
        break
      end
      sync()
    end
    $ 1522 "Direction: Base Z+"
    global move_thread_flag_1522=0
    thread move_thread_1522():
      enter_critical
      move_thread_flag_1522 = 1
      local towardsPos=calculate_point_to_move_towards(p[0.0,0.0,0.0,0.0,0.0,0.0], [0.0,0.0,1.0], 0.08)
      movel(towardsPos, a=0.15, v=0.1)
      move_thread_flag_1522 = 2
      exit_critical
    end
    move_thread_flag_1522 = 0
    move_thread_han_1522 = run move_thread_1522()
    while (True):
      sleep(1.0E-10)
      if (move_thread_flag_1522 > 1):
        join move_thread_han_1522
        $ 1523 "Until (distance)"
        break
      end
      sync()
    end
    $ 1524 "Linea12_B" "breakAfter"
    movel(Linea12_B_p, a=0.5, v=0.1)
    $ 1525 "bajada_comprobacion"
    $ 1526 "Direction: Base Z-"
    global move_thread_flag_1526=0
    thread move_thread_1526():
      enter_critical
      move_thread_flag_1526 = 1
      local towardsPos=calculate_point_to_move_towards(p[0.0,0.0,0.0,0.0,0.0,0.0], [0.0,0.0,-1.0], 0.071)
      movel(towardsPos, a=0.15, v=0.1)
      move_thread_flag_1526 = 2
      exit_critical
    end
    move_thread_flag_1526 = 0
    move_thread_han_1526 = run move_thread_1526()
    while (True):
      sleep(1.0E-10)
      if (move_thread_flag_1526 > 1):
        join move_thread_han_1526
        $ 1527 "Until (distance)"
        break
      end
      sync()
    end
    $ 1528 "Direction: Base Z-"
    global move_thread_flag_1528=0
    thread move_thread_1528():
      enter_critical
      move_thread_flag_1528 = 1
      local towardsPos=calculate_point_to_move_towards(p[0.0,0.0,0.0,0.0,0.0,0.0], [0.0,0.0,-1.0], 1000.0)
      movel(towardsPos, a=0.007, v=0.007)
      move_thread_flag_1528 = 2
      exit_critical
    end
    move_thread_flag_1528 = 0
    move_thread_han_1528 = run move_thread_1528()
    while (True):
      local targetTcpDirection=get_target_tcp_speed()
      local stepsToRetract=tool_contact(direction=targetTcpDirection)
      if (stepsToRetract > 0):
        kill move_thread_han_1528
        stopl(0.02)
        local backTrackMovement=get_actual_joint_positions_history(stepsToRetract)
        local contactPose=get_forward_kin(backTrackMovement)
        local posDir=[targetTcpDirection[0],targetTcpDirection[1],targetTcpDirection[2]]
        local retractTo=contactPose
        if (norm(posDir) > 1e-6):
          local normalizedPosDir=normalize(posDir)
          local additionalRetraction=p[normalizedPosDir[0] * 0.0, normalizedPosDir[1] * 0.0, normalizedPosDir[2] * 0.0, 0, 0, 0]
          retractTo = pose_sub(contactPose, additionalRetraction)
        end
        movel(retractTo, a=0.02, v=0.1)
        $ 1529 "Until (tool_contact_detection)"
        break
      end
      sync()
    end
    $ 1530 "Direction: Base Z+"
    global move_thread_flag_1530=0
    thread move_thread_1530():
      enter_critical
      move_thread_flag_1530 = 1
      local towardsPos=calculate_point_to_move_towards(p[0.0,0.0,0.0,0.0,0.0,0.0], [0.0,0.0,1.0], 0.08)
      movel(towardsPos, a=0.15, v=0.1)
      move_thread_flag_1530 = 2
      exit_critical
    end
    move_thread_flag_1530 = 0
    move_thread_han_1530 = run move_thread_1530()
    while (True):
      sleep(1.0E-10)
      if (move_thread_flag_1530 > 1):
        join move_thread_han_1530
        $ 1531 "Until (distance)"
        break
      end
      sync()
    end
    $ 1532 "AB"
    $ 1533 "'desbaste_inicial'"
    # 'desbaste_inicial'
    $ 1534 "bajada_broca≔p[0,0,-0.008,0,0,0]"
    global bajada_broca=p[0,0,-0.008,0,0,0]
    $ 1535 "barrenos_menos1≔7"
    global barrenos_menos1=7
    $ 1536 "barreno_actual≔0"
    global barreno_actual=0
    $ 1537 "Loop barreno_actual≤barrenos_menos1"
    while (barreno_actual <= barrenos_menos1):
      $ 1538 "Perforacion"
      $ 1539 "MoveL"
      $ 1540 "If barreno_actual≟2"
      if (barreno_actual == 2):
        $ 1541 "barreno_actual≔barreno_actual+1"
        global barreno_actual=barreno_actual+1
      end
      $ 1542 "internos≔interpolate_pose(Linea12_A, Linea12_B, barreno_actual/barrenos_menos1)"
      global internos= interpolate_pose (Linea12_A_p, Linea12_B_p, barreno_actual/barrenos_menos1)
      $ 1543 "internos" "breakAfter"
      movel(internos, a=0.5, v=0.1)
      $ 1544 "'desbaste_inicial'"
      # 'desbaste_inicial'
      $ 1545 "bajada_broca≔p[0,0,-0.024,0,0,0]"
      global bajada_broca=p[0,0,-0.024,0,0,0]
      $ 1546 "bajada≔p[0,0,0.024,0,0,0]"
      global bajada=p[0,0,0.024,0,0,0]
      $ 1547 "Direction: Base Z-"
      global move_thread_flag_1547=0
      thread move_thread_1547():
        enter_critical
        move_thread_flag_1547 = 1
        local towardsPos=calculate_point_to_move_towards(p[0.0,0.0,0.0,0.0,0.0,0.0], [0.0,0.0,-1.0], 0.071)
        movel(towardsPos, a=0.15, v=0.1)
        move_thread_flag_1547 = 2
        exit_critical
      end
      move_thread_flag_1547 = 0
      move_thread_han_1547 = run move_thread_1547()
      while (True):
        sleep(1.0E-10)
        if (move_thread_flag_1547 > 1):
          join move_thread_han_1547
          $ 1548 "Until (distance)"
          break
        end
        sync()
      end
      $ 1549 "Direction: Base Z-"
      global move_thread_flag_1549=0
      thread move_thread_1549():
        enter_critical
        move_thread_flag_1549 = 1
        local towardsPos=calculate_point_to_move_towards(p[0.0,0.0,0.0,0.0,0.0,0.0], [0.0,0.0,-1.0], 1000.0)
        movel(towardsPos, a=0.007, v=0.007)
        move_thread_flag_1549 = 2
        exit_critical
      end
      move_thread_flag_1549 = 0
      move_thread_han_1549 = run move_thread_1549()
      while (True):
        local targetTcpDirection=get_target_tcp_speed()
        local stepsToRetract=tool_contact(direction=targetTcpDirection)
        if (stepsToRetract > 0):
          kill move_thread_han_1549
          stopl(0.02)
          local backTrackMovement=get_actual_joint_positions_history(stepsToRetract)
          local contactPose=get_forward_kin(backTrackMovement)
          local posDir=[targetTcpDirection[0],targetTcpDirection[1],targetTcpDirection[2]]
          local retractTo=contactPose
          if (norm(posDir) > 1e-6):
            local normalizedPosDir=normalize(posDir)
            local additionalRetraction=p[normalizedPosDir[0] * 0.0, normalizedPosDir[1] * 0.0, normalizedPosDir[2] * 0.0, 0, 0, 0]
            retractTo = pose_sub(contactPose, additionalRetraction)
          end
          movel(retractTo, a=0.02, v=0.1)
          $ 1550 "Until (tool_contact_detection)"
          break
        end
        sync()
      end
      $ 1551 "Popup: punto contacto alanzdo"
      popup("punto contacto alanzdo", "Mensaje", False, False, blocking=True)
      $ 1552 "Direction: Base Z+"
      global move_thread_flag_1552=0
      thread move_thread_1552():
        enter_critical
        move_thread_flag_1552 = 1
        local towardsPos=calculate_point_to_move_towards(p[0.0,0.0,0.0,0.0,0.0,0.0], [0.0,0.0,1.0], 0.002)
        movel(towardsPos, a=0.015, v=0.015)
        move_thread_flag_1552 = 2
        exit_critical
      end
      move_thread_flag_1552 = 0
      move_thread_han_1552 = run move_thread_1552()
      while (True):
        sleep(1.0E-10)
        if (move_thread_flag_1552 > 1):
          join move_thread_han_1552
          $ 1553 "Until (distance)"
          break
        end
        sync()
      end
      $ 1554 "Wait: 0.3"
      sleep(0.3)
      $ 1555 "Set CO[1]=Encender"
      set_configurable_digital_out(1, True)
      $ 1556 "Wait: 0.3"
      sleep(0.3)
      $ 1557 "Loop 1 times"
      Loop_126 = 0
      while (Loop_126 < 1):
        $ 1558 "bajar≔pose_add(get_actual_tcp_pose(), bajada_broca)"
        global bajar= pose_add ( get_actual_tcp_pose (), bajada_broca)
        $ 1559 "bajar" "breakAfter"
        movel(bajar, a=0.004, v=0.004)
        $ 1560 "subir≔pose_sub(get_actual_tcp_pose(), bajada_broca)"
        global subir= pose_sub ( get_actual_tcp_pose (), bajada_broca)
        $ 1561 "Direction: Base Z+"
        global move_thread_flag_1561=0
        thread move_thread_1561():
          enter_critical
          move_thread_flag_1561 = 1
          local towardsPos=calculate_point_to_move_towards(p[0.0,0.0,0.0,0.0,0.0,0.0], [0.0,0.0,1.0], 0.002)
          movel(towardsPos, a=0.015, v=0.015)
          move_thread_flag_1561 = 2
          exit_critical
        end
        move_thread_flag_1561 = 0
        move_thread_han_1561 = run move_thread_1561()
        while (True):
          sleep(1.0E-10)
          if (move_thread_flag_1561 > 1):
            join move_thread_han_1561
            $ 1562 "Until (distance)"
            break
          end
          sync()
        end
        $ 1563 "Set CO[1]=Apagar"
        set_configurable_digital_out(1, False)
        $ 1564 "subir" "breakAfter"
        movel(subir, a=0.015, v=0.015)
        $ 1565 "bajada_broca≔pose_sub(bajada_broca, bajada)"
        global bajada_broca= pose_sub (bajada_broca, bajada)
        Loop_126 = Loop_126 + 1
      end
      $ 1566 "Direction: Base Z+"
      global move_thread_flag_1566=0
      thread move_thread_1566():
        enter_critical
        move_thread_flag_1566 = 1
        local towardsPos=calculate_point_to_move_towards(p[0.0,0.0,0.0,0.0,0.0,0.0], [0.0,0.0,1.0], 0.08)
        movel(towardsPos, a=0.15, v=0.1)
        move_thread_flag_1566 = 2
        exit_critical
      end
      move_thread_flag_1566 = 0
      move_thread_han_1566 = run move_thread_1566()
      while (True):
        sleep(1.0E-10)
        if (move_thread_flag_1566 > 1):
          join move_thread_han_1566
          $ 1567 "Until (distance)"
          break
        end
        sync()
      end
      $ 1568 "Set CO[1]=Apagar"
      set_configurable_digital_out(1, False)
      $ 1569 "barreno_actual≔barreno_actual+1"
      global barreno_actual=barreno_actual+1
    end
    $ 1572 "Popup: Linea12 con chica Terminada!"
    popup("Linea12 con chica Terminada!", "Mensaje", False, False, blocking=True)
    $ 1573 "Linea13"
    $ 1574 "Marcar_puntos"
    $ 1575 "MoveL"
    $ 1576 "Linea13_A" "breakAfter"
    movel(Linea13_A_p, a=0.5, v=0.1)
    $ 1577 "bajada_comprobacion"
    $ 1578 "Direction: Base Z-"
    global move_thread_flag_1578=0
    thread move_thread_1578():
      enter_critical
      move_thread_flag_1578 = 1
      local towardsPos=calculate_point_to_move_towards(p[0.0,0.0,0.0,0.0,0.0,0.0], [0.0,0.0,-1.0], 0.071)
      movel(towardsPos, a=0.15, v=0.1)
      move_thread_flag_1578 = 2
      exit_critical
    end
    move_thread_flag_1578 = 0
    move_thread_han_1578 = run move_thread_1578()
    while (True):
      sleep(1.0E-10)
      if (move_thread_flag_1578 > 1):
        join move_thread_han_1578
        $ 1579 "Until (distance)"
        break
      end
      sync()
    end
    $ 1580 "Direction: Base Z-"
    global move_thread_flag_1580=0
    thread move_thread_1580():
      enter_critical
      move_thread_flag_1580 = 1
      local towardsPos=calculate_point_to_move_towards(p[0.0,0.0,0.0,0.0,0.0,0.0], [0.0,0.0,-1.0], 1000.0)
      movel(towardsPos, a=0.007, v=0.007)
      move_thread_flag_1580 = 2
      exit_critical
    end
    move_thread_flag_1580 = 0
    move_thread_han_1580 = run move_thread_1580()
    while (True):
      local targetTcpDirection=get_target_tcp_speed()
      local stepsToRetract=tool_contact(direction=targetTcpDirection)
      if (stepsToRetract > 0):
        kill move_thread_han_1580
        stopl(0.02)
        local backTrackMovement=get_actual_joint_positions_history(stepsToRetract)
        local contactPose=get_forward_kin(backTrackMovement)
        local posDir=[targetTcpDirection[0],targetTcpDirection[1],targetTcpDirection[2]]
        local retractTo=contactPose
        if (norm(posDir) > 1e-6):
          local normalizedPosDir=normalize(posDir)
          local additionalRetraction=p[normalizedPosDir[0] * 0.0, normalizedPosDir[1] * 0.0, normalizedPosDir[2] * 0.0, 0, 0, 0]
          retractTo = pose_sub(contactPose, additionalRetraction)
        end
        movel(retractTo, a=0.02, v=0.1)
        $ 1581 "Until (tool_contact_detection)"
        break
      end
      sync()
    end
    $ 1582 "Direction: Base Z+"
    global move_thread_flag_1582=0
    thread move_thread_1582():
      enter_critical
      move_thread_flag_1582 = 1
      local towardsPos=calculate_point_to_move_towards(p[0.0,0.0,0.0,0.0,0.0,0.0], [0.0,0.0,1.0], 0.08)
      movel(towardsPos, a=0.15, v=0.1)
      move_thread_flag_1582 = 2
      exit_critical
    end
    move_thread_flag_1582 = 0
    move_thread_han_1582 = run move_thread_1582()
    while (True):
      sleep(1.0E-10)
      if (move_thread_flag_1582 > 1):
        join move_thread_han_1582
        $ 1583 "Until (distance)"
        break
      end
      sync()
    end
    $ 1584 "Linea13_B" "breakAfter"
    movel(Linea13_B_p, a=0.5, v=0.1)
    $ 1585 "bajada_comprobacion"
    $ 1586 "Direction: Base Z-"
    global move_thread_flag_1586=0
    thread move_thread_1586():
      enter_critical
      move_thread_flag_1586 = 1
      local towardsPos=calculate_point_to_move_towards(p[0.0,0.0,0.0,0.0,0.0,0.0], [0.0,0.0,-1.0], 0.071)
      movel(towardsPos, a=0.15, v=0.1)
      move_thread_flag_1586 = 2
      exit_critical
    end
    move_thread_flag_1586 = 0
    move_thread_han_1586 = run move_thread_1586()
    while (True):
      sleep(1.0E-10)
      if (move_thread_flag_1586 > 1):
        join move_thread_han_1586
        $ 1587 "Until (distance)"
        break
      end
      sync()
    end
    $ 1588 "Direction: Base Z-"
    global move_thread_flag_1588=0
    thread move_thread_1588():
      enter_critical
      move_thread_flag_1588 = 1
      local towardsPos=calculate_point_to_move_towards(p[0.0,0.0,0.0,0.0,0.0,0.0], [0.0,0.0,-1.0], 1000.0)
      movel(towardsPos, a=0.007, v=0.007)
      move_thread_flag_1588 = 2
      exit_critical
    end
    move_thread_flag_1588 = 0
    move_thread_han_1588 = run move_thread_1588()
    while (True):
      local targetTcpDirection=get_target_tcp_speed()
      local stepsToRetract=tool_contact(direction=targetTcpDirection)
      if (stepsToRetract > 0):
        kill move_thread_han_1588
        stopl(0.02)
        local backTrackMovement=get_actual_joint_positions_history(stepsToRetract)
        local contactPose=get_forward_kin(backTrackMovement)
        local posDir=[targetTcpDirection[0],targetTcpDirection[1],targetTcpDirection[2]]
        local retractTo=contactPose
        if (norm(posDir) > 1e-6):
          local normalizedPosDir=normalize(posDir)
          local additionalRetraction=p[normalizedPosDir[0] * 0.0, normalizedPosDir[1] * 0.0, normalizedPosDir[2] * 0.0, 0, 0, 0]
          retractTo = pose_sub(contactPose, additionalRetraction)
        end
        movel(retractTo, a=0.02, v=0.1)
        $ 1589 "Until (tool_contact_detection)"
        break
      end
      sync()
    end
    $ 1590 "Direction: Base Z+"
    global move_thread_flag_1590=0
    thread move_thread_1590():
      enter_critical
      move_thread_flag_1590 = 1
      local towardsPos=calculate_point_to_move_towards(p[0.0,0.0,0.0,0.0,0.0,0.0], [0.0,0.0,1.0], 0.08)
      movel(towardsPos, a=0.15, v=0.1)
      move_thread_flag_1590 = 2
      exit_critical
    end
    move_thread_flag_1590 = 0
    move_thread_han_1590 = run move_thread_1590()
    while (True):
      sleep(1.0E-10)
      if (move_thread_flag_1590 > 1):
        join move_thread_han_1590
        $ 1591 "Until (distance)"
        break
      end
      sync()
    end
    $ 1592 "AB"
    $ 1593 "'desbaste_inicial'"
    # 'desbaste_inicial'
    $ 1594 "bajada_broca≔p[0,0,-0.008,0,0,0]"
    global bajada_broca=p[0,0,-0.008,0,0,0]
    $ 1595 "barrenos_menos1≔2"
    global barrenos_menos1=2
    $ 1596 "barreno_actual≔0"
    global barreno_actual=0
    $ 1597 "Loop barreno_actual≤barrenos_menos1"
    while (barreno_actual <= barrenos_menos1):
      $ 1598 "Perforacion"
      $ 1599 "MoveL"
      $ 1602 "internos≔interpolate_pose(Linea13_A, Linea13_B, barreno_actual/barrenos_menos1)"
      global internos= interpolate_pose (Linea13_A_p, Linea13_B_p, barreno_actual/barrenos_menos1)
      $ 1603 "internos" "breakAfter"
      movel(internos, a=0.5, v=0.1)
      $ 1604 "'desbaste_inicial'"
      # 'desbaste_inicial'
      $ 1605 "bajada_broca≔p[0,0,-0.024,0,0,0]"
      global bajada_broca=p[0,0,-0.024,0,0,0]
      $ 1606 "bajada≔p[0,0,0.024,0,0,0]"
      global bajada=p[0,0,0.024,0,0,0]
      $ 1607 "Direction: Base Z-"
      global move_thread_flag_1607=0
      thread move_thread_1607():
        enter_critical
        move_thread_flag_1607 = 1
        local towardsPos=calculate_point_to_move_towards(p[0.0,0.0,0.0,0.0,0.0,0.0], [0.0,0.0,-1.0], 0.071)
        movel(towardsPos, a=0.15, v=0.1)
        move_thread_flag_1607 = 2
        exit_critical
      end
      move_thread_flag_1607 = 0
      move_thread_han_1607 = run move_thread_1607()
      while (True):
        sleep(1.0E-10)
        if (move_thread_flag_1607 > 1):
          join move_thread_han_1607
          $ 1608 "Until (distance)"
          break
        end
        sync()
      end
      $ 1609 "Direction: Base Z-"
      global move_thread_flag_1609=0
      thread move_thread_1609():
        enter_critical
        move_thread_flag_1609 = 1
        local towardsPos=calculate_point_to_move_towards(p[0.0,0.0,0.0,0.0,0.0,0.0], [0.0,0.0,-1.0], 1000.0)
        movel(towardsPos, a=0.007, v=0.007)
        move_thread_flag_1609 = 2
        exit_critical
      end
      move_thread_flag_1609 = 0
      move_thread_han_1609 = run move_thread_1609()
      while (True):
        local targetTcpDirection=get_target_tcp_speed()
        local stepsToRetract=tool_contact(direction=targetTcpDirection)
        if (stepsToRetract > 0):
          kill move_thread_han_1609
          stopl(0.02)
          local backTrackMovement=get_actual_joint_positions_history(stepsToRetract)
          local contactPose=get_forward_kin(backTrackMovement)
          local posDir=[targetTcpDirection[0],targetTcpDirection[1],targetTcpDirection[2]]
          local retractTo=contactPose
          if (norm(posDir) > 1e-6):
            local normalizedPosDir=normalize(posDir)
            local additionalRetraction=p[normalizedPosDir[0] * 0.0, normalizedPosDir[1] * 0.0, normalizedPosDir[2] * 0.0, 0, 0, 0]
            retractTo = pose_sub(contactPose, additionalRetraction)
          end
          movel(retractTo, a=0.02, v=0.1)
          $ 1610 "Until (tool_contact_detection)"
          break
        end
        sync()
      end
      $ 1611 "Popup: punto contacto alanzdo"
      popup("punto contacto alanzdo", "Mensaje", False, False, blocking=True)
      $ 1612 "Direction: Base Z+"
